C07321=1123.386,90.409,-56.038,-179.966,7.860,149.482
C07322=1123.381,90.658,-56.056,-179.965,7.864,149.482
C07323=1123.376,90.907,-56.074,-179.963,7.868,149.483
C07324=1123.371,91.156,-56.092,-179.961,7.872,149.483
C07325=1123.366,91.406,-56.111,-179.960,7.876,149.484
C07326=1123.362,91.655,-56.129,-179.958,7.879,149.484
C07327=1123.357,91.904,-56.147,-179.957,7.883,149.484
C07328=1123.352,92.153,-56.165,-179.956,7.886,149.485
C07329=1123.347,92.403,-56.183,-179.954,7.891,149.486
C07330=1123.343,92.652,-56.202,-179.953,7.895,149.486
C07331=1123.337,92.902,-56.220,-179.951,7.898,149.486
C07332=1123.332,93.150,-56.239,-179.950,7.902,149.487
C07333=1123.327,93.400,-56.257,-179.948,7.906,149.487
C07334=1123.323,93.650,-56.275,-179.946,7.910,149.488
C07335=1123.318,93.899,-56.293,-179.945,7.914,149.488
C07336=1123.313,94.148,-56.312,-179.943,7.918,149.489
C07337=1123.308,94.397,-56.331,-179.942,7.922,149.489
C07338=1123.304,94.647,-56.349,-179.939,7.926,149.489
C07339=1123.299,94.896,-56.367,-179.938,7.930,149.490
C07340=1123.293,95.145,-56.386,-179.936,7.934,149.490
C07341=1123.289,95.395,-56.404,-179.934,7.938,149.491
C07342=1123.284,95.644,-56.422,-179.933,7.942,149.491
C07343=1123.280,95.892,-56.441,-179.931,7.946,149.491
C07344=1123.274,96.142,-56.460,-179.929,7.949,149.492
C07345=1123.270,96.392,-56.478,-179.928,7.953,149.492
C07346=1123.265,96.640,-56.497,-179.926,7.957,149.493
C07347=1123.259,96.890,-56.515,-179.925,7.961,149.493
C07348=1123.255,97.140,-56.534,-179.923,7.965,149.493
C07349=1123.250,97.388,-56.552,-179.921,7.969,149.494
C07350=1123.245,97.638,-56.571,-179.919,7.973,149.494
C07351=1123.241,97.887,-56.590,-179.917,7.977,149.495
C07352=1123.236,98.136,-56.608,-179.916,7.981,149.495
C07353=1123.230,98.386,-56.627,-179.913,7.984,149.495
C07354=1123.226,98.635,-56.646,-179.912,7.988,149.496
C07355=1123.221,98.884,-56.664,-179.910,7.992,149.496
C07356=1123.216,99.133,-56.683,-179.908,7.997,149.497
C07357=1123.212,99.383,-56.701,-179.906,8.000,149.497
C07358=1123.206,99.632,-56.721,-179.904,8.004,149.497
C07359=1123.202,99.881,-56.739,-179.903,8.008,149.498
C07360=1123.197,100.130,-56.758,-179.901,8.012,149.498
C07361=1123.192,100.379,-56.777,-179.898,8.016,149.498
C07362=1123.188,100.629,-56.795,-179.896,8.020,149.498
C07363=1123.182,100.878,-56.815,-179.895,8.024,149.499
C07364=1123.178,101.127,-56.833,-179.893,8.028,149.499
C07365=1123.173,101.376,-56.852,-179.891,8.031,149.500
C07366=1123.168,101.626,-56.870,-179.889,8.036,149.500
C07367=1123.163,101.875,-56.890,-179.887,8.039,149.500
C07368=1123.158,102.124,-56.908,-179.885,8.043,149.501
C07369=1123.153,102.374,-56.927,-179.883,8.047,149.501
C07370=1123.150,102.588,-56.944,-179.882,8.051,149.501
C07371=1123.145,102.802,-56.960,-179.880,8.054,149.502
C07372=1123.141,103.016,-56.976,-179.878,8.058,149.502
C07373=1123.136,103.232,-56.992,-179.877,8.061,149.502
C07374=1123.133,103.446,-57.009,-179.874,8.064,149.502
C07375=1123.129,103.661,-57.025,-179.872,8.068,149.503
C07376=1123.125,103.875,-57.042,-179.871,8.070,149.503
C07377=1123.120,104.089,-57.058,-179.869,8.074,149.503
C07378=1123.115,104.339,-57.077,-179.867,8.078,149.503
C07379=1123.111,104.588,-57.096,-179.865,8.082,149.504
C07380=1123.106,104.838,-57.116,-179.863,8.086,149.504
C07381=1123.101,105.086,-57.134,-179.861,8.089,149.504
C07382=1123.096,105.336,-57.153,-179.858,8.094,149.505
C07383=1123.092,105.585,-57.172,-179.857,8.098,149.505
C07384=1123.087,105.834,-57.192,-179.855,8.101,149.505
C07385=1123.081,106.083,-57.211,-179.852,8.105,149.505
C07386=1123.077,106.333,-57.230,-179.850,8.109,149.506
C07387=1123.072,106.581,-57.249,-179.848,8.114,149.506
C07388=1123.067,106.831,-57.269,-179.846,8.117,149.506
C07389=1123.062,107.080,-57.287,-179.844,8.121,149.507
C07390=1123.058,107.330,-57.306,-179.841,8.125,149.507
C07391=1123.052,107.579,-57.326,-179.839,8.128,149.507
C07392=1123.048,107.828,-57.345,-179.837,8.132,149.507
C07393=1123.044,108.077,-57.364,-179.834,8.137,149.508
C07394=1123.038,108.326,-57.384,-179.832,8.140,149.508
C07395=1123.033,108.576,-57.403,-179.830,8.144,149.508
C07396=1123.029,108.824,-57.422,-179.828,8.148,149.508
C07397=1123.024,109.074,-57.442,-179.825,8.152,149.508
C07398=1123.019,109.324,-57.461,-179.823,8.156,149.509
C07399=1123.015,109.572,-57.480,-179.821,8.159,149.509
C07400=1123.010,109.822,-57.500,-179.818,8.163,149.509
C07401=1123.005,110.071,-57.519,-179.816,8.167,149.509
C07402=1123.000,110.320,-57.539,-179.813,8.171,149.510
C07403=1122.995,110.570,-57.558,-179.811,8.175,149.510
C07404=1122.991,110.818,-57.577,-179.809,8.179,149.510
C07405=1122.986,111.067,-57.597,-179.807,8.182,149.510
C07406=1122.981,111.317,-57.617,-179.805,8.186,149.510
C07407=1122.976,111.566,-57.636,-179.803,8.190,149.511
C07408=1122.971,111.815,-57.656,-179.801,8.193,149.511
C07409=1122.967,112.065,-57.676,-179.799,8.197,149.511
C07410=1122.962,112.313,-57.694,-179.797,8.200,149.512
C07411=1122.957,112.563,-57.714,-179.796,8.203,149.512
C07412=1122.953,112.812,-57.734,-179.794,8.207,149.512
C07413=1122.947,113.061,-57.754,-179.792,8.210,149.512
C07414=1122.943,113.310,-57.773,-179.790,8.214,149.513
C07415=1122.938,113.560,-57.793,-179.788,8.218,149.513
C07416=1122.933,113.809,-57.812,-179.786,8.221,149.513
C07417=1122.928,114.058,-57.833,-179.784,8.225,149.514
C07418=1122.923,114.307,-57.852,-179.782,8.228,149.514
C07419=1122.918,114.556,-57.872,-179.781,8.231,149.514
C07420=1122.913,114.806,-57.891,-179.779,8.235,149.514
C07421=1122.910,115.054,-57.911,-179.777,8.238,149.515
C07422=1122.905,115.304,-57.931,-179.775,8.242,149.515
C07423=1122.900,115.553,-57.950,-179.773,8.245,149.515
C07424=1122.895,115.802,-57.970,-179.771,8.249,149.516
C07425=1122.890,116.051,-57.990,-179.769,8.253,149.516
C07426=1122.886,116.266,-58.007,-179.767,8.256,149.516
C07427=1122.882,116.480,-58.025,-179.766,8.258,149.516
C07428=1122.878,116.695,-58.041,-179.765,8.261,149.516
C07429=1122.873,116.908,-58.059,-179.763,8.264,149.517
C07430=1122.869,117.123,-58.076,-179.761,8.267,149.517
C07431=1122.865,117.338,-58.092,-179.760,8.270,149.517
C07432=1122.861,117.552,-58.110,-179.758,8.273,149.517
C07433=1122.857,117.767,-58.127,-179.756,8.276,149.518
C07434=1122.852,118.016,-58.147,-179.755,8.280,149.518
C07435=1122.847,118.265,-58.167,-179.753,8.283,149.518
C07436=1122.842,118.514,-58.187,-179.751,8.286,149.518
C07437=1122.838,118.763,-58.207,-179.749,8.290,149.519
C07438=1122.833,119.012,-58.227,-179.747,8.293,149.519
C07439=1122.829,119.262,-58.247,-179.745,8.297,149.519
C07440=1122.824,119.511,-58.266,-179.744,8.300,149.520
C07441=1122.819,119.760,-58.287,-179.742,8.303,149.520
C07442=1122.814,120.008,-58.307,-179.740,8.307,149.520
C07443=1122.810,120.258,-58.326,-179.738,8.310,149.520
C07444=1122.805,120.507,-58.347,-179.737,8.313,149.521
C07445=1122.800,120.757,-58.366,-179.735,8.317,149.521
C07446=1122.796,121.005,-58.387,-179.733,8.320,149.521
C07447=1122.790,121.255,-58.407,-179.730,8.324,149.521
C07448=1122.785,121.504,-58.427,-179.729,8.327,149.522
C07449=1122.781,121.753,-58.447,-179.727,8.330,149.522
C07450=1122.776,122.002,-58.467,-179.725,8.334,149.522
C07451=1122.772,122.251,-58.487,-179.723,8.337,149.522
C07452=1122.767,122.501,-58.507,-179.722,8.340,149.523
C07453=1122.762,122.750,-58.528,-179.720,8.344,149.523
C07454=1122.757,122.999,-58.548,-179.718,8.348,149.523
C07455=1122.753,123.248,-58.568,-179.716,8.351,149.524
C07456=1122.748,123.497,-58.588,-179.715,8.354,149.524
C07457=1122.743,123.746,-58.608,-179.713,8.357,149.524
C07458=1122.738,123.995,-58.628,-179.711,8.361,149.524
C07459=1122.733,124.244,-58.649,-179.709,8.364,149.525
C07460=1122.729,124.493,-58.669,-179.707,8.367,149.525
C07461=1122.724,124.742,-58.690,-179.705,8.371,149.525
C07462=1122.720,124.992,-58.709,-179.704,8.375,149.526
C07463=1122.715,125.241,-58.730,-179.702,8.377,149.526
C07464=1122.710,125.490,-58.751,-179.700,8.381,149.526
C07465=1122.706,125.739,-58.771,-179.698,8.384,149.526
C07466=1122.701,125.989,-58.791,-179.697,8.388,149.527
C07467=1122.696,126.238,-58.812,-179.695,8.391,149.527
C07468=1122.691,126.487,-58.832,-179.693,8.395,149.527
C07469=1122.687,126.736,-58.852,-179.692,8.397,149.527
C07470=1122.682,126.985,-58.873,-179.690,8.401,149.528
C07471=1122.676,127.234,-58.893,-179.688,8.405,149.528
C07472=1122.672,127.483,-58.913,-179.686,8.407,149.528
C07473=1122.667,127.732,-58.933,-179.684,8.411,149.528
C07474=1122.662,127.981,-58.954,-179.682,8.414,149.529
C07475=1122.658,128.230,-58.975,-179.681,8.417,149.529
C07476=1122.653,128.479,-58.996,-179.679,8.421,149.529
C07477=1122.648,128.728,-59.016,-179.677,8.424,149.530
C07478=1122.644,128.977,-59.036,-179.676,8.427,149.530
C07479=1122.639,129.226,-59.057,-179.674,8.431,149.530
C07480=1122.634,129.475,-59.078,-179.672,8.434,149.530
C07481=1122.629,129.725,-59.097,-179.671,8.437,149.531
C07482=1122.625,129.940,-59.116,-179.669,8.440,149.531
C07483=1122.621,130.154,-59.134,-179.668,8.444,149.531
C07484=1122.617,130.368,-59.151,-179.666,8.446,149.532
C07485=1122.614,130.583,-59.169,-179.665,8.449,149.532
C07486=1122.609,130.797,-59.187,-179.663,8.452,149.532
C07487=1122.605,131.011,-59.205,-179.662,8.455,149.532
C07488=1122.601,131.226,-59.222,-179.660,8.457,149.532
C07489=1122.597,131.439,-59.240,-179.659,8.460,149.533
C07490=1122.592,131.689,-59.261,-179.657,8.464,149.533
C07491=1122.587,131.938,-59.281,-179.655,8.467,149.533
C07492=1122.582,132.187,-59.302,-179.654,8.470,149.534
C07493=1122.578,132.436,-59.322,-179.652,8.474,149.534
C07494=1122.573,132.686,-59.344,-179.651,8.477,149.534
C07495=1122.569,132.935,-59.364,-179.649,8.480,149.534
C07496=1122.564,133.183,-59.386,-179.646,8.484,149.535
C07497=1122.559,133.432,-59.406,-179.645,8.487,149.535
C07498=1122.554,133.682,-59.427,-179.643,8.490,149.535
C07499=1122.550,133.931,-59.448,-179.642,8.493,149.536
C07500=1122.545,134.180,-59.469,-179.640,8.497,149.536
C07501=1122.540,134.429,-59.489,-179.638,8.500,149.536
C07502=1122.535,134.678,-59.510,-179.637,8.503,149.536
C07503=1122.531,134.926,-59.531,-179.635,8.507,149.537
C07504=1122.526,135.176,-59.552,-179.634,8.510,149.537
C07505=1122.522,135.425,-59.573,-179.632,8.513,149.537
C07506=1122.517,135.675,-59.594,-179.630,8.517,149.538
C07507=1122.512,135.923,-59.614,-179.629,8.520,149.538
C07508=1122.507,136.172,-59.636,-179.627,8.524,149.538
C07509=1122.502,136.421,-59.657,-179.625,8.526,149.539
C07510=1122.498,136.670,-59.677,-179.623,8.530,149.539
C07511=1122.493,136.920,-59.698,-179.622,8.534,149.539
C07512=1122.489,137.169,-59.719,-179.620,8.536,149.539
C07513=1122.484,137.418,-59.740,-179.619,8.540,149.540
C07514=1122.479,137.667,-59.761,-179.617,8.543,149.540
C07515=1122.474,137.916,-59.782,-179.615,8.546,149.540
C07516=1122.469,138.165,-59.803,-179.614,8.550,149.541
C07517=1122.465,138.414,-59.824,-179.612,8.553,149.541
C07518=1122.460,138.664,-59.845,-179.610,8.557,149.541
C07519=1122.456,138.912,-59.867,-179.609,8.560,149.542
C07520=1122.451,139.161,-59.887,-179.607,8.564,149.542
C07521=1122.446,139.410,-59.909,-179.606,8.566,149.542
C07522=1122.441,139.659,-59.930,-179.604,8.570,149.543
C07523=1122.437,139.909,-59.951,-179.603,8.573,149.543
C07524=1122.432,140.157,-59.972,-179.601,8.576,149.543
C07525=1122.427,140.407,-59.993,-179.600,8.579,149.544
C07526=1122.423,140.655,-60.014,-179.598,8.583,149.544
C07527=1122.418,140.904,-60.035,-179.596,8.587,149.544
C07528=1122.413,141.154,-60.057,-179.595,8.589,149.545
C07529=1122.408,141.403,-60.078,-179.593,8.593,149.545
C07530=1122.404,141.652,-60.099,-179.592,8.596,149.545
C07531=1122.399,141.900,-60.120,-179.590,8.600,149.546
C07532=1122.395,142.150,-60.142,-179.589,8.603,149.546
C07533=1122.390,142.399,-60.163,-179.587,8.606,149.546
C07534=1122.385,142.648,-60.184,-179.586,8.610,149.547
C07535=1122.380,142.897,-60.205,-179.584,8.613,149.547
C07536=1122.376,143.147,-60.227,-179.583,8.616,149.547
C07537=1122.371,143.395,-60.248,-179.581,8.620,149.548
C07538=1122.367,143.610,-60.266,-179.580,8.623,149.548
C07539=1122.363,143.823,-60.285,-179.578,8.625,149.548
C07540=1122.359,144.038,-60.303,-179.577,8.628,149.549
C07541=1122.355,144.252,-60.322,-179.576,8.631,149.549
C07542=1122.351,144.466,-60.340,-179.574,8.634,149.549
C07543=1122.347,144.681,-60.359,-179.573,8.637,149.550
C07544=1122.343,144.895,-60.376,-179.572,8.640,149.550
C07545=1122.339,145.109,-60.395,-179.570,8.642,149.550
C07546=1122.334,145.359,-60.416,-179.568,8.647,149.550
C07547=1122.329,145.607,-60.438,-179.566,8.650,149.551
C07548=1122.324,145.856,-60.460,-179.563,8.654,149.551
C07549=1122.321,146.105,-60.481,-179.561,8.658,149.551
C07550=1122.316,146.354,-60.502,-179.558,8.662,149.551
C07551=1122.311,146.603,-60.524,-179.556,8.666,149.552
C07552=1122.306,146.853,-60.545,-179.553,8.670,149.552
C07553=1122.301,147.101,-60.567,-179.551,8.673,149.552
C07554=1122.297,147.350,-60.589,-179.548,8.677,149.552
C07555=1122.292,147.600,-60.610,-179.546,8.681,149.552
C07556=1122.287,147.849,-60.632,-179.543,8.685,149.552
C07557=1122.282,148.097,-60.653,-179.541,8.689,149.553
C07558=1122.278,148.347,-60.675,-179.538,8.693,149.553
C07559=1122.273,148.595,-60.697,-179.536,8.696,149.553
C07560=1122.268,148.844,-60.718,-179.533,8.700,149.553
C07561=1122.264,149.093,-60.740,-179.531,8.704,149.553
C07562=1122.260,149.342,-60.761,-179.529,8.707,149.554
C07563=1122.255,149.591,-60.783,-179.526,8.712,149.554
C07564=1122.250,149.840,-60.805,-179.524,8.715,149.554
C07565=1122.245,150.089,-60.827,-179.521,8.719,149.554
C07566=1122.240,150.339,-60.849,-179.519,8.722,149.554
C07567=1122.235,150.588,-60.870,-179.517,8.726,149.555
C07568=1122.231,150.837,-60.892,-179.514,8.730,149.555
C07569=1122.226,151.086,-60.914,-179.512,8.733,149.555
C07570=1122.222,151.335,-60.936,-179.510,8.737,149.555
C07571=1122.217,151.584,-60.958,-179.506,8.741,149.555
C07572=1122.212,151.832,-60.979,-179.504,8.744,149.555
C07573=1122.208,152.082,-61.001,-179.502,8.748,149.556
C07574=1122.203,152.330,-61.023,-179.499,8.751,149.556
C07575=1122.199,152.580,-61.045,-179.497,8.755,149.556
C07576=1122.194,152.828,-61.067,-179.495,8.758,149.556
C07577=1122.190,153.078,-61.089,-179.492,8.762,149.556
C07578=1122.184,153.327,-61.111,-179.490,8.766,149.556
C07579=1122.180,153.576,-61.133,-179.487,8.769,149.556
C07580=1122.175,153.824,-61.155,-179.485,8.772,149.557
C07581=1122.171,154.074,-61.177,-179.483,8.776,149.557
C07582=1122.166,154.322,-61.199,-179.480,8.780,149.557
C07583=1122.162,154.571,-61.221,-179.478,8.783,149.557
C07584=1122.156,154.820,-61.244,-179.475,8.786,149.557
C07585=1122.152,155.069,-61.266,-179.473,8.790,149.557
C07586=1122.147,155.318,-61.287,-179.471,8.793,149.557
C07587=1122.143,155.567,-61.309,-179.468,8.797,149.558
C07588=1122.138,155.816,-61.331,-179.465,8.800,149.558
C07589=1122.133,156.065,-61.354,-179.463,8.804,149.558
C07590=1122.129,156.314,-61.377,-179.461,8.807,149.558
C07591=1122.124,156.563,-61.398,-179.459,8.810,149.558
C07592=1122.120,156.812,-61.420,-179.456,8.814,149.558
C07593=1122.115,157.061,-61.443,-179.454,8.818,149.559
C07594=1122.111,157.275,-61.462,-179.452,8.820,149.559
C07595=1122.107,157.489,-61.481,-179.449,8.823,149.559
C07596=1122.103,157.703,-61.500,-179.448,8.826,149.559
C07597=1122.099,157.917,-61.519,-179.445,8.829,149.559
C07598=1122.095,158.131,-61.538,-179.444,8.832,149.559
C07599=1122.091,158.346,-61.557,-179.441,8.835,149.559
C07600=1122.087,158.560,-61.577,-179.439,8.837,149.559
C07601=1122.084,158.774,-61.596,-179.437,8.841,149.559
C07602=1122.078,159.023,-61.619,-179.435,8.844,149.559
C07603=1122.074,159.272,-61.641,-179.433,8.847,149.560
C07604=1122.069,159.520,-61.663,-179.430,8.850,149.560
C07605=1122.064,159.770,-61.686,-179.428,8.853,149.560
C07606=1122.060,160.019,-61.709,-179.425,8.857,149.560
C07607=1122.055,160.267,-61.730,-179.423,8.860,149.560
C07608=1122.050,160.517,-61.753,-179.421,8.864,149.560
C07609=1122.046,160.766,-61.776,-179.418,8.867,149.560
C07610=1122.041,161.014,-61.797,-179.416,8.870,149.560
C07611=1122.037,161.263,-61.821,-179.414,8.873,149.561
C07612=1122.032,161.513,-61.843,-179.411,8.876,149.561
C07613=1122.027,161.761,-61.866,-179.409,8.880,149.561
C07614=1122.023,162.010,-61.888,-179.407,8.883,149.561
C07615=1122.019,162.259,-61.911,-179.404,8.886,149.561
C07616=1122.014,162.509,-61.933,-179.402,8.890,149.561
C07617=1122.009,162.757,-61.956,-179.399,8.893,149.561
C07618=1122.004,163.006,-61.978,-179.397,8.896,149.561
C07619=1122.000,163.255,-62.001,-179.395,8.899,149.561
C07620=1121.995,163.504,-62.024,-179.392,8.902,149.561
C07621=1121.991,163.753,-62.046,-179.390,8.905,149.561
C07622=1121.986,164.002,-62.069,-179.388,8.909,149.562
C07623=1121.982,164.251,-62.091,-179.385,8.912,149.562
C07624=1121.977,164.500,-62.114,-179.383,8.915,149.562
C07625=1121.973,164.748,-62.137,-179.381,8.919,149.562
C07626=1121.968,164.998,-62.160,-179.378,8.922,149.562
C07627=1121.964,165.247,-62.183,-179.376,8.924,149.562
C07628=1121.958,165.495,-62.206,-179.374,8.928,149.562
C07629=1121.954,165.744,-62.228,-179.372,8.931,149.562
C07630=1121.949,165.993,-62.251,-179.369,8.934,149.562
C07631=1121.945,166.242,-62.274,-179.367,8.937,149.563
C07632=1121.940,166.490,-62.297,-179.364,8.940,149.563
C07633=1121.935,166.740,-62.319,-179.362,8.944,149.563
C07634=1121.931,166.989,-62.342,-179.359,8.947,149.563
C07635=1121.926,167.238,-62.366,-179.358,8.949,149.563
C07636=1121.922,167.487,-62.389,-179.355,8.952,149.563
C07637=1121.917,167.736,-62.411,-179.353,8.956,149.563
C07638=1121.912,167.985,-62.434,-179.351,8.959,149.563
C07639=1121.908,168.233,-62.457,-179.348,8.962,149.563
C07640=1121.903,168.482,-62.480,-179.346,8.965,149.563
C07641=1121.899,168.731,-62.503,-179.344,8.968,149.564
C07642=1121.894,168.979,-62.526,-179.342,8.971,149.564
C07643=1121.889,169.229,-62.548,-179.339,8.974,149.564
C07644=1121.885,169.478,-62.572,-179.337,8.977,149.564
C07645=1121.880,169.727,-62.595,-179.335,8.981,149.564
C07646=1121.876,169.976,-62.618,-179.333,8.983,149.564
C07647=1121.871,170.225,-62.641,-179.330,8.986,149.564
C07648=1121.866,170.473,-62.664,-179.328,8.990,149.564
C07649=1121.862,170.722,-62.687,-179.326,8.993,149.564
C07650=1121.858,170.936,-62.708,-179.324,8.995,149.564
C07651=1121.854,171.151,-62.727,-179.322,8.997,149.564
C07652=1121.850,171.364,-62.747,-179.320,9.000,149.565
C07653=1121.846,171.578,-62.767,-179.318,9.003,149.565
C07654=1121.842,171.792,-62.787,-179.316,9.006,149.565
C07655=1121.838,172.007,-62.806,-179.314,9.008,149.565
C07656=1121.834,172.220,-62.827,-179.313,9.011,149.565
C07657=1121.830,172.434,-62.847,-179.310,9.014,149.565
C07658=1121.825,172.683,-62.870,-179.308,9.016,149.565
C07659=1121.821,172.932,-62.893,-179.306,9.019,149.565
C07660=1121.817,173.181,-62.916,-179.304,9.023,149.565
C07661=1121.812,173.430,-62.939,-179.302,9.025,149.565
C07662=1121.807,173.679,-62.963,-179.299,9.028,149.565
C07663=1121.803,173.928,-62.986,-179.297,9.032,149.566
C07664=1121.798,174.177,-63.009,-179.295,9.035,149.566
C07665=1121.793,174.426,-63.033,-179.293,9.037,149.566
C07666=1121.790,174.674,-63.056,-179.290,9.040,149.566
C07667=1121.785,174.923,-63.080,-179.288,9.044,149.566
C07668=1121.780,175.172,-63.103,-179.286,9.046,149.566
C07669=1121.775,175.421,-63.126,-179.284,9.049,149.566
C07670=1121.771,175.670,-63.150,-179.282,9.053,149.566
C07671=1121.766,175.919,-63.173,-179.280,9.055,149.566
C07672=1121.762,176.168,-63.197,-179.277,9.058,149.566
C07673=1121.758,176.416,-63.220,-179.275,9.061,149.566
C07674=1121.753,176.665,-63.243,-179.273,9.064,149.567
C07675=1121.748,176.914,-63.267,-179.271,9.067,149.567
C07676=1121.744,177.163,-63.291,-179.269,9.070,149.567
C07677=1121.739,177.412,-63.314,-179.267,9.073,149.567
C07678=1121.734,177.661,-63.337,-179.264,9.076,149.567
C07679=1121.730,177.910,-63.361,-179.263,9.079,149.567
C07680=1121.725,178.158,-63.385,-179.260,9.082,149.567
C07681=1121.721,178.407,-63.408,-179.258,9.085,149.567
C07682=1121.716,178.656,-63.432,-179.256,9.087,149.567
C07683=1121.712,178.905,-63.456,-179.254,9.091,149.567
C07684=1121.707,179.154,-63.479,-179.252,9.093,149.568
C07685=1121.702,179.403,-63.502,-179.249,9.097,149.568
C07686=1121.698,179.651,-63.526,-179.246,9.100,149.568
C07687=1121.693,179.900,-63.550,-179.244,9.103,149.568
C07688=1121.688,180.149,-63.573,-179.241,9.106,149.568
C07689=1121.684,180.398,-63.597,-179.238,9.110,149.568
C07690=1121.679,180.647,-63.621,-179.235,9.113,149.568
C07691=1121.675,180.895,-63.645,-179.233,9.116,149.568
C07692=1121.670,181.144,-63.668,-179.230,9.119,149.568
C07693=1121.666,181.393,-63.692,-179.227,9.123,149.568
C07694=1121.662,181.642,-63.716,-179.224,9.126,149.568
C07695=1121.657,181.891,-63.740,-179.222,9.129,149.568
C07696=1121.653,182.140,-63.763,-179.219,9.132,149.568
C07697=1121.648,182.388,-63.787,-179.216,9.135,149.568
C07698=1121.644,182.637,-63.811,-179.214,9.138,149.568
C07699=1121.639,182.886,-63.835,-179.211,9.141,149.568
C07700=1121.634,183.135,-63.859,-179.209,9.144,149.568
C07701=1121.629,183.383,-63.883,-179.206,9.147,149.568
C07702=1121.625,183.632,-63.906,-179.204,9.150,149.568
C07703=1121.621,183.882,-63.931,-179.201,9.154,149.568
C07704=1121.616,184.130,-63.955,-179.198,9.156,149.568
C07705=1121.612,184.379,-63.978,-179.196,9.159,149.568
C07706=1121.608,184.592,-63.999,-179.193,9.162,149.568
C07707=1121.604,184.807,-64.020,-179.191,9.165,149.568
C07708=1121.600,185.020,-64.040,-179.189,9.167,149.568
C07709=1121.596,185.234,-64.061,-179.187,9.170,149.568
C07710=1121.592,185.448,-64.082,-179.185,9.173,149.568
C07711=1121.588,185.663,-64.102,-179.183,9.175,149.568
C07712=1121.584,185.876,-64.123,-179.180,9.178,149.568
C07713=1121.580,186.090,-64.144,-179.178,9.180,149.568
C07714=1121.576,186.339,-64.168,-179.176,9.183,149.568
C07715=1121.572,186.587,-64.192,-179.174,9.185,149.568
C07716=1121.566,186.837,-64.216,-179.171,9.189,149.568
C07717=1121.562,187.086,-64.240,-179.169,9.192,149.568
C07718=1121.558,187.334,-64.264,-179.167,9.194,149.568
C07719=1121.553,187.583,-64.289,-179.164,9.197,149.568
C07720=1121.548,187.832,-64.312,-179.162,9.200,149.568
C07721=1121.544,188.080,-64.336,-179.160,9.203,149.568
C07722=1121.540,188.329,-64.361,-179.157,9.206,149.568
C07723=1121.535,188.578,-64.385,-179.155,9.209,149.568
C07724=1121.530,188.826,-64.410,-179.153,9.211,149.568
C07725=1121.526,189.075,-64.434,-179.150,9.214,149.568
C07726=1121.521,189.325,-64.458,-179.148,9.217,149.568
C07727=1121.517,189.573,-64.482,-179.146,9.220,149.569
C07728=1121.512,189.822,-64.506,-179.144,9.222,149.569
C07729=1121.507,190.070,-64.531,-179.141,9.225,149.569
C07730=1121.504,190.320,-64.555,-179.140,9.227,149.569
C07731=1121.498,190.568,-64.580,-179.137,9.230,149.569
C07732=1121.494,190.817,-64.604,-179.135,9.233,149.569
C07733=1121.490,191.066,-64.628,-179.133,9.236,149.569
C07734=1121.485,191.315,-64.653,-179.131,9.239,149.569
C07735=1121.481,191.563,-64.677,-179.129,9.242,149.569
C07736=1121.476,191.812,-64.702,-179.127,9.244,149.569
C07737=1121.472,192.061,-64.726,-179.125,9.246,149.569
C07738=1121.467,192.309,-64.750,-179.122,9.250,149.569
C07739=1121.462,192.558,-64.775,-179.121,9.252,149.569
C07740=1121.458,192.807,-64.799,-179.119,9.255,149.569
C07741=1121.453,193.056,-64.824,-179.116,9.258,149.569
C07742=1121.449,193.304,-64.848,-179.115,9.260,149.570
C07743=1121.444,193.554,-64.873,-179.113,9.263,149.570
C07744=1121.440,193.802,-64.897,-179.111,9.265,149.570
C07745=1121.435,194.051,-64.922,-179.109,9.268,149.570
C07746=1121.431,194.300,-64.946,-179.107,9.271,149.570
C07747=1121.426,194.549,-64.971,-179.105,9.273,149.570
C07748=1121.422,194.797,-64.995,-179.104,9.276,149.570
C07749=1121.418,195.046,-65.020,-179.101,9.279,149.570
C07750=1121.413,195.294,-65.045,-179.100,9.282,149.571
C07751=1121.409,195.543,-65.069,-179.098,9.284,149.571
C07752=1121.404,195.792,-65.094,-179.096,9.287,149.571
C07753=1121.399,196.041,-65.119,-179.095,9.289,149.571
C07754=1121.395,196.290,-65.143,-179.093,9.292,149.571
C07755=1121.390,196.539,-65.168,-179.090,9.296,149.571
C07756=1121.386,196.787,-65.192,-179.086,9.299,149.571
C07757=1121.381,197.036,-65.218,-179.083,9.303,149.571
C07758=1121.377,197.284,-65.242,-179.080,9.307,149.571
C07759=1121.372,197.534,-65.267,-179.077,9.309,149.571
C07760=1121.368,197.782,-65.291,-179.073,9.313,149.571
C07761=1121.363,198.030,-65.316,-179.070,9.317,149.571
C07762=1121.360,198.244,-65.338,-179.067,9.319,149.571
C07763=1121.356,198.458,-65.359,-179.064,9.322,149.571
C07764=1121.352,198.673,-65.380,-179.061,9.325,149.571
C07765=1121.348,198.886,-65.401,-179.059,9.328,149.570
C07766=1121.344,199.100,-65.423,-179.056,9.331,149.570
C07767=1121.341,199.314,-65.444,-179.053,9.334,149.570
C07768=1121.336,199.527,-65.465,-179.050,9.337,149.570
C07769=1121.332,199.741,-65.487,-179.047,9.339,149.570
C07770=1121.329,199.990,-65.512,-179.045,9.342,149.570
C07771=1121.323,200.239,-65.537,-179.041,9.346,149.570
C07772=1121.319,200.487,-65.563,-179.038,9.349,149.570
C07773=1121.315,200.736,-65.587,-179.035,9.352,149.570
C07774=1121.310,200.985,-65.612,-179.032,9.355,149.570
C07775=1121.305,201.233,-65.637,-179.028,9.358,149.569
C07776=1121.302,201.482,-65.662,-179.025,9.362,149.569
C07777=1121.297,201.731,-65.687,-179.023,9.364,149.569
C07778=1121.292,201.980,-65.712,-179.019,9.368,149.569
C07779=1121.287,202.228,-65.738,-179.016,9.371,149.569
C07780=1121.284,202.477,-65.763,-179.013,9.373,149.569
C07781=1121.279,202.725,-65.787,-179.009,9.377,149.569
C07782=1121.275,202.974,-65.813,-179.007,9.380,149.569
C07783=1121.269,203.223,-65.838,-179.004,9.383,149.569
C07784=1121.265,203.472,-65.864,-179.001,9.385,149.568
C07785=1121.261,203.721,-65.888,-178.997,9.389,149.568
C07786=1121.257,203.969,-65.913,-178.994,9.392,149.568
C07787=1121.252,204.218,-65.939,-178.992,9.395,149.568
C07788=1121.247,204.466,-65.964,-178.989,9.398,149.568
C07789=1121.243,204.715,-65.990,-178.986,9.400,149.568
C07790=1121.238,204.963,-66.015,-178.983,9.403,149.568
C07791=1121.234,205.213,-66.040,-178.981,9.406,149.568
C07792=1121.229,205.462,-66.066,-178.978,9.409,149.568
C07793=1121.225,205.709,-66.090,-178.975,9.412,149.568
C07794=1121.221,205.958,-66.116,-178.972,9.414,149.567
C07795=1121.216,206.207,-66.141,-178.969,9.417,149.567
C07796=1121.212,206.456,-66.167,-178.966,9.420,149.567
C07797=1121.208,206.704,-66.192,-178.964,9.423,149.567
C07798=1121.203,206.953,-66.218,-178.961,9.426,149.567
C07799=1121.199,207.201,-66.244,-178.958,9.429,149.567
C07800=1121.194,207.451,-66.269,-178.955,9.432,149.567
C07801=1121.189,207.699,-66.294,-178.952,9.435,149.567
C07802=1121.185,207.948,-66.320,-178.950,9.438,149.567
C07803=1121.181,208.196,-66.345,-178.947,9.440,149.567
C07804=1121.176,208.445,-66.371,-178.945,9.443,149.567
C07805=1121.172,208.693,-66.397,-178.942,9.446,149.567
C07806=1121.167,208.942,-66.422,-178.939,9.449,149.567
C07807=1121.163,209.190,-66.448,-178.937,9.451,149.567
C07808=1121.158,209.440,-66.473,-178.935,9.454,149.567
C07809=1121.154,209.689,-66.499,-178.932,9.457,149.567
C07810=1121.149,209.937,-66.524,-178.929,9.460,149.567
C07811=1121.145,210.185,-66.550,-178.927,9.463,149.567
C07812=1121.141,210.434,-66.575,-178.925,9.465,149.567
C07813=1121.136,210.683,-66.601,-178.922,9.468,149.567
C07814=1121.132,210.931,-66.627,-178.919,9.471,149.567
C07815=1121.127,211.180,-66.652,-178.917,9.473,149.567
C07816=1121.122,211.429,-66.679,-178.915,9.476,149.567
C07817=1121.118,211.678,-66.704,-178.912,9.479,149.567
C07818=1121.114,211.890,-66.726,-178.910,9.482,149.567
C07819=1121.110,212.104,-66.749,-178.909,9.484,149.567
C07820=1121.107,212.318,-66.770,-178.907,9.486,149.567
C07821=1121.103,212.532,-66.793,-178.905,9.489,149.567
C07822=1121.099,212.746,-66.815,-178.903,9.491,149.567
C07823=1121.096,212.959,-66.837,-178.901,9.493,149.567
C07824=1121.092,213.173,-66.860,-178.899,9.496,149.567
C07825=1121.088,213.387,-66.881,-178.898,9.498,149.567
C07826=1121.083,213.636,-66.908,-178.895,9.502,149.568
C07827=1121.079,213.884,-66.934,-178.893,9.504,149.568
C07828=1121.074,214.132,-66.959,-178.891,9.507,149.568
C07829=1121.070,214.381,-66.985,-178.889,9.510,149.568
C07830=1121.066,214.630,-67.011,-178.887,9.512,149.568
C07831=1121.061,214.879,-67.037,-178.885,9.516,149.568
C07832=1121.057,215.128,-67.063,-178.883,9.518,149.568
C07833=1121.052,215.375,-67.089,-178.881,9.521,149.568
C07834=1121.048,215.624,-67.115,-178.879,9.524,149.569
C07835=1121.044,215.873,-67.141,-178.877,9.527,149.569
C07836=1121.039,216.122,-67.167,-178.875,9.530,149.569
C07837=1121.035,216.370,-67.193,-178.873,9.533,149.569
C07838=1121.031,216.619,-67.219,-178.870,9.536,149.569
C07839=1121.026,216.867,-67.245,-178.868,9.539,149.569
C07840=1121.021,217.116,-67.271,-178.866,9.541,149.569
C07841=1121.017,217.364,-67.297,-178.864,9.545,149.569
C07842=1121.013,217.613,-67.323,-178.861,9.548,149.569
C07843=1121.008,217.862,-67.349,-178.860,9.550,149.570
C07844=1121.004,218.110,-67.376,-178.857,9.554,149.570
C07845=1121.000,218.359,-67.402,-178.855,9.557,149.570
C07846=1120.995,218.607,-67.427,-178.852,9.560,149.570
C07847=1120.990,218.856,-67.454,-178.850,9.563,149.570
C07848=1120.986,219.104,-67.480,-178.848,9.566,149.570
C07849=1120.982,219.353,-67.506,-178.846,9.569,149.570
C07850=1120.978,219.601,-67.532,-178.843,9.572,149.570
C07851=1120.973,219.851,-67.558,-178.841,9.575,149.570
C07852=1120.969,220.099,-67.585,-178.838,9.578,149.570
C07853=1120.964,220.348,-67.611,-178.836,9.581,149.570
C07854=1120.960,220.596,-67.638,-178.833,9.585,149.571
C07855=1120.956,220.845,-67.663,-178.831,9.588,149.571
C07856=1120.950,221.093,-67.690,-178.828,9.591,149.571
C07857=1120.946,221.341,-67.716,-178.826,9.594,149.571
C07858=1120.942,221.590,-67.743,-178.823,9.597,149.571
C07859=1120.937,221.839,-67.769,-178.821,9.600,149.571
C07860=1120.933,222.087,-67.795,-178.818,9.603,149.571
C07861=1120.928,222.336,-67.822,-178.816,9.606,149.571
C07862=1120.925,222.584,-67.848,-178.813,9.609,149.571
C07863=1120.920,222.833,-67.874,-178.811,9.613,149.571
C07864=1120.916,223.082,-67.901,-178.807,9.616,149.571
C07865=1120.911,223.330,-67.928,-178.805,9.619,149.571
C07866=1120.907,223.579,-67.954,-178.802,9.622,149.571
C07867=1120.902,223.827,-67.981,-178.800,9.625,149.571
C07868=1120.898,224.076,-68.007,-178.797,9.629,149.571
C07869=1120.893,224.325,-68.034,-178.794,9.632,149.572
C07870=1120.889,224.573,-68.060,-178.791,9.635,149.571
C07871=1120.885,224.821,-68.087,-178.788,9.638,149.571
C07872=1120.880,225.070,-68.113,-178.786,9.641,149.572
C07873=1120.876,225.319,-68.140,-178.782,9.645,149.571
C07874=1120.872,225.532,-68.163,-178.780,9.647,149.571
C07875=1120.868,225.746,-68.185,-178.778,9.650,149.572
C07876=1120.865,225.959,-68.208,-178.775,9.653,149.571
C07877=1120.861,226.173,-68.232,-178.772,9.656,149.571
C07878=1120.857,226.387,-68.254,-178.770,9.659,149.572
C07879=1120.853,226.600,-68.277,-178.768,9.661,149.571
C07880=1120.849,226.813,-68.301,-178.765,9.664,149.571
C07881=1120.845,227.027,-68.323,-178.762,9.667,149.571
C07882=1120.841,227.275,-68.350,-178.759,9.670,149.571
C07883=1120.837,227.524,-68.377,-178.756,9.674,149.571
C07884=1120.833,227.772,-68.403,-178.753,9.677,149.571
C07885=1120.828,228.021,-68.430,-178.750,9.680,149.571
C07886=1120.824,228.270,-68.457,-178.747,9.683,149.571
C07887=1120.820,228.518,-68.484,-178.744,9.687,149.571
C07888=1120.815,228.767,-68.511,-178.741,9.690,149.571
C07889=1120.811,229.015,-68.538,-178.737,9.693,149.571
C07890=1120.807,229.264,-68.564,-178.734,9.696,149.571
C07891=1120.802,229.512,-68.591,-178.731,9.700,149.571
C07892=1120.797,229.761,-68.618,-178.728,9.702,149.571
C07893=1120.793,230.009,-68.645,-178.724,9.706,149.570
C07894=1120.789,230.257,-68.672,-178.721,9.709,149.570
C07895=1120.785,230.506,-68.699,-178.718,9.712,149.570
C07896=1120.780,230.755,-68.726,-178.715,9.715,149.570
C07897=1120.775,231.003,-68.753,-178.711,9.719,149.570
C07898=1120.772,231.252,-68.780,-178.709,9.721,149.570
C07899=1120.767,231.500,-68.807,-178.705,9.725,149.570
C07900=1120.762,231.749,-68.834,-178.702,9.728,149.570
C07901=1120.759,231.997,-68.862,-178.699,9.730,149.570
C07902=1120.754,232.246,-68.889,-178.695,9.734,149.570
C07903=1120.750,232.494,-68.916,-178.693,9.737,149.569
C07904=1120.745,232.742,-68.943,-178.690,9.739,149.569
C07905=1120.741,232.991,-68.970,-178.687,9.742,149.569
C07906=1120.737,233.240,-68.997,-178.684,9.745,149.569
C07907=1120.732,233.488,-69.025,-178.681,9.748,149.569
C07908=1120.728,233.736,-69.052,-178.677,9.751,149.569
C07909=1120.723,233.985,-69.079,-178.674,9.754,149.569
C07910=1120.720,234.234,-69.106,-178.671,9.757,149.569
C07911=1120.715,234.482,-69.134,-178.668,9.760,149.568
C07912=1120.711,234.730,-69.161,-178.665,9.762,149.568
C07913=1120.706,234.979,-69.188,-178.662,9.765,149.568
C07914=1120.702,235.228,-69.215,-178.660,9.768,149.568
C07915=1120.698,235.476,-69.243,-178.657,9.771,149.568
C07916=1120.693,235.724,-69.270,-178.655,9.773,149.568
C07917=1120.688,235.973,-69.297,-178.652,9.776,149.568
C07918=1120.684,236.221,-69.325,-178.649,9.778,149.568
C07919=1120.680,236.470,-69.352,-178.646,9.781,149.568
C07920=1120.675,236.718,-69.380,-178.643,9.784,149.568
C07921=1120.671,236.967,-69.408,-178.640,9.787,149.567
C07922=1120.667,237.215,-69.435,-178.638,9.789,149.567
C07923=1120.662,237.463,-69.462,-178.635,9.792,149.567
C07924=1120.658,237.712,-69.490,-178.632,9.794,149.567
C07925=1120.654,237.960,-69.518,-178.630,9.796,149.567
C07926=1120.647,238.351,-69.560,-178.626,9.801,149.567
C07927=1120.640,238.744,-69.604,-178.621,9.805,149.567
C07928=1120.633,239.136,-69.648,-178.618,9.809,149.567
C07929=1120.627,239.526,-69.691,-178.614,9.813,149.567
C07930=1120.622,239.811,-69.723,-178.611,9.816,149.567
C07931=1120.617,240.094,-69.754,-178.608,9.818,149.566
C07932=1120.612,240.378,-69.786,-178.605,9.821,149.567
C07933=1120.607,240.661,-69.817,-178.602,9.824,149.566
C07934=1120.603,240.910,-69.845,-178.600,9.827,149.566
C07935=1120.598,241.158,-69.872,-178.597,9.829,149.566
C07936=1120.593,241.407,-69.901,-178.596,9.832,149.566
C07937=1120.589,241.656,-69.928,-178.593,9.834,149.566
C07938=1120.585,241.904,-69.956,-178.591,9.837,149.566
C07939=1120.581,242.152,-69.984,-178.588,9.839,149.566
C07940=1120.576,242.401,-70.011,-178.586,9.841,149.566
C07941=1120.572,242.649,-70.039,-178.585,9.843,149.566
C07942=1120.568,242.897,-70.067,-178.582,9.846,149.566
C07943=1120.563,243.145,-70.096,-178.580,9.848,149.566
C07944=1120.559,243.395,-70.123,-178.578,9.851,149.566
C07945=1120.555,243.642,-70.151,-178.576,9.853,149.566
C07946=1120.550,243.890,-70.179,-178.574,9.855,149.566
C07947=1120.546,244.139,-70.206,-178.571,9.858,149.566
C07948=1120.541,244.388,-70.234,-178.569,9.860,149.566
C07949=1120.538,244.636,-70.262,-178.567,9.863,149.566
C07950=1120.533,244.884,-70.290,-178.565,9.865,149.567
C07951=1120.529,245.133,-70.318,-178.564,9.867,149.567
C07952=1120.525,245.381,-70.345,-178.562,9.870,149.567
C07953=1120.520,245.630,-70.374,-178.560,9.872,149.567
C07954=1120.516,245.878,-70.402,-178.558,9.874,149.567
C07955=1120.512,246.126,-70.430,-178.556,9.877,149.567
C07956=1120.507,246.375,-70.458,-178.554,9.880,149.567
C07957=1120.502,246.623,-70.486,-178.553,9.882,149.567
C07958=1120.499,246.872,-70.514,-178.551,9.884,149.567
C07959=1120.494,247.120,-70.541,-178.549,9.887,149.567
C07960=1120.490,247.369,-70.570,-178.547,9.889,149.568
C07961=1120.486,247.616,-70.598,-178.544,9.893,149.567
C07962=1120.482,247.865,-70.626,-178.538,9.897,149.567
C07963=1120.477,248.113,-70.654,-178.533,9.902,149.567
C07964=1120.473,248.362,-70.683,-178.528,9.905,149.566
C07965=1120.469,248.610,-70.710,-178.523,9.910,149.566
C07966=1120.464,248.858,-70.739,-178.518,9.914,149.566
C07967=1120.460,249.106,-70.767,-178.513,9.918,149.565
C07968=1120.456,249.355,-70.795,-178.508,9.922,149.565
C07969=1120.452,249.604,-70.824,-178.504,9.925,149.565
C07970=1120.447,249.852,-70.852,-178.500,9.929,149.564
C07971=1120.443,250.101,-70.880,-178.496,9.932,149.564
C07972=1120.438,250.348,-70.908,-178.492,9.935,149.564
C07973=1120.434,250.597,-70.937,-178.488,9.938,149.564
C07974=1120.430,250.846,-70.965,-178.484,9.941,149.563
C07975=1120.425,251.094,-70.993,-178.481,9.944,149.563
C07976=1120.422,251.342,-71.022,-178.477,9.947,149.563
C07977=1120.416,251.590,-71.051,-178.473,9.950,149.563
C07978=1120.413,251.839,-71.079,-178.470,9.953,149.562
C07979=1120.408,252.088,-71.107,-178.467,9.955,149.562
C07980=1120.404,252.335,-71.136,-178.464,9.958,149.562
C07981=1120.400,252.584,-71.165,-178.462,9.960,149.562
C07982=1120.396,252.797,-71.188,-178.459,9.962,149.562
C07983=1120.392,253.010,-71.213,-178.457,9.964,149.562
C07984=1120.389,253.224,-71.238,-178.455,9.966,149.562
C07985=1120.385,253.437,-71.262,-178.454,9.967,149.562
C07986=1120.382,253.650,-71.287,-178.452,9.969,149.562
C07987=1120.378,253.864,-71.312,-178.450,9.971,149.561
C07988=1120.374,254.077,-71.336,-178.449,9.972,149.561
C07989=1120.370,254.291,-71.360,-178.448,9.974,149.561
C07990=1120.366,254.538,-71.389,-178.445,9.976,149.561
C07991=1120.362,254.787,-71.418,-178.444,9.978,149.562
C07992=1120.357,255.036,-71.446,-178.443,9.979,149.562
C07993=1120.353,255.283,-71.475,-178.442,9.981,149.562
C07994=1120.349,255.532,-71.504,-178.442,9.982,149.562
C07995=1120.345,255.780,-71.532,-178.440,9.983,149.562
C07996=1120.340,256.028,-71.561,-178.439,9.985,149.562
C07997=1120.336,256.277,-71.590,-178.437,9.988,149.562
C07998=1120.332,256.525,-71.618,-178.434,9.991,149.562
C07999=1120.328,256.774,-71.647,-178.431,9.994,149.562
C08000=1120.323,257.021,-71.676,-178.428,9.997,149.562
C08001=1120.319,257.270,-71.704,-178.425,10.000,149.562
C08002=1120.315,257.519,-71.733,-178.422,10.002,149.562
C08003=1120.310,257.766,-71.762,-178.420,10.005,149.562
C08004=1120.306,258.015,-71.790,-178.417,10.008,149.562
C08005=1120.302,258.263,-71.820,-178.414,10.011,149.562
C08006=1120.298,258.512,-71.849,-178.411,10.014,149.561
C08007=1120.294,258.759,-71.877,-178.408,10.016,149.561
C08008=1120.289,259.008,-71.906,-178.405,10.019,149.561
C08009=1120.285,259.256,-71.935,-178.402,10.022,149.561
C08010=1120.280,259.505,-71.964,-178.399,10.025,149.561
C08011=1120.276,259.753,-71.992,-178.396,10.028,149.561
C08012=1120.272,260.001,-72.022,-178.393,10.031,149.561
C08013=1120.268,260.250,-72.051,-178.390,10.034,149.561
C08014=1120.264,260.498,-72.080,-178.387,10.036,149.561
C08015=1120.260,260.745,-72.109,-178.384,10.039,149.561
C08016=1120.255,260.994,-72.137,-178.380,10.042,149.560
C08017=1120.251,261.242,-72.167,-178.377,10.045,149.560
C08018=1120.247,261.491,-72.196,-178.374,10.048,149.560
C08019=1120.242,261.740,-72.225,-178.370,10.051,149.560
C08020=1120.239,261.988,-72.254,-178.367,10.054,149.560
C08021=1120.234,262.235,-72.283,-178.364,10.057,149.560
C08022=1120.229,262.484,-72.312,-178.361,10.060,149.559
C08023=1120.225,262.732,-72.341,-178.358,10.063,149.559
C08024=1120.221,262.981,-72.371,-178.354,10.065,149.559
C08025=1120.217,263.229,-72.400,-178.351,10.069,149.559
C08026=1120.212,263.478,-72.429,-178.347,10.071,149.559
C08027=1120.208,263.725,-72.457,-178.344,10.074,149.559
C08028=1120.204,263.973,-72.487,-178.340,10.077,149.558
C08029=1120.200,264.221,-72.516,-178.337,10.080,149.558
C08030=1120.196,264.470,-72.546,-178.333,10.083,149.558
C08031=1120.192,264.718,-72.575,-178.331,10.085,149.558
C08032=1120.187,264.966,-72.605,-178.328,10.088,149.558
C08033=1120.183,265.215,-72.633,-178.326,10.090,149.558
C08034=1120.179,265.463,-72.663,-178.323,10.093,149.557
C08035=1120.174,265.711,-72.692,-178.320,10.095,149.557
C08036=1120.170,265.959,-72.721,-178.318,10.097,149.557
C08037=1120.166,266.208,-72.751,-178.315,10.100,149.557
C08038=1120.162,266.421,-72.776,-178.312,10.102,149.557
C08039=1120.159,266.634,-72.802,-178.311,10.104,149.557
C08040=1120.155,266.847,-72.827,-178.308,10.106,149.557
C08041=1120.151,267.060,-72.852,-178.306,10.108,149.557
C08042=1120.148,267.273,-72.877,-178.304,10.110,149.557
C08043=1120.144,267.487,-72.902,-178.301,10.112,149.557
C08044=1120.141,267.700,-72.928,-178.299,10.115,149.557
C08045=1120.137,267.913,-72.953,-178.296,10.117,149.557
C08046=1120.133,268.161,-72.983,-178.294,10.119,149.556
C08047=1120.129,268.409,-73.012,-178.291,10.122,149.556
C08048=1120.125,268.658,-73.042,-178.288,10.125,149.556
C08049=1120.120,268.906,-73.072,-178.286,10.127,149.556
C08050=1120.116,269.155,-73.101,-178.283,10.130,149.556
C08051=1120.111,269.402,-73.130,-178.280,10.132,149.556
C08052=1120.107,269.650,-73.160,-178.278,10.134,149.556
C08053=1120.103,269.898,-73.190,-178.275,10.137,149.556
C08054=1120.098,270.146,-73.219,-178.272,10.140,149.556
C08055=1120.094,270.395,-73.249,-178.269,10.143,149.555
C08056=1120.090,270.643,-73.278,-178.266,10.145,149.555
C08057=1120.086,270.891,-73.308,-178.264,10.147,149.555
C08058=1120.081,271.140,-73.338,-178.261,10.150,149.555
C08059=1120.078,271.388,-73.368,-178.258,10.153,149.555
C08060=1120.074,271.636,-73.398,-178.255,10.156,149.555
C08061=1120.069,271.885,-73.427,-178.252,10.158,149.555
C08062=1120.065,272.133,-73.457,-178.249,10.161,149.555
C08063=1120.061,272.380,-73.487,-178.246,10.163,149.554
C08064=1120.056,272.629,-73.517,-178.243,10.166,149.554
C08065=1120.052,272.877,-73.546,-178.240,10.168,149.554
C08066=1120.048,273.125,-73.576,-178.238,10.171,149.554
C08067=1120.044,273.373,-73.606,-178.235,10.174,149.554
C08068=1120.040,273.622,-73.635,-178.232,10.177,149.554
C08069=1120.035,273.869,-73.666,-178.229,10.179,149.554
C08070=1120.031,274.118,-73.696,-178.226,10.182,149.554
C08071=1120.027,274.366,-73.725,-178.222,10.185,149.553
C08072=1120.023,274.614,-73.755,-178.220,10.187,149.553
C08073=1120.018,274.862,-73.785,-178.217,10.190,149.553
C08074=1120.014,275.110,-73.815,-178.214,10.193,149.553
C08075=1120.011,275.359,-73.845,-178.211,10.196,149.553
C08076=1120.006,275.607,-73.876,-178.207,10.198,149.553
C08077=1120.002,275.855,-73.905,-178.204,10.201,149.553
C08078=1119.998,276.103,-73.936,-178.201,10.204,149.553
C08079=1119.993,276.351,-73.966,-178.199,10.206,149.552
C08080=1119.989,276.599,-73.996,-178.195,10.209,149.552
C08081=1119.985,276.847,-74.025,-178.192,10.212,149.552
C08082=1119.981,277.096,-74.056,-178.189,10.214,149.552
C08083=1119.977,277.344,-74.086,-178.186,10.217,149.552
C08084=1119.973,277.592,-74.116,-178.183,10.219,149.552
C08085=1119.968,277.840,-74.146,-178.180,10.222,149.551
C08086=1119.964,278.088,-74.176,-178.177,10.225,149.551
C08087=1119.960,278.336,-74.206,-178.174,10.227,149.551
C08088=1119.956,278.585,-74.237,-178.171,10.230,149.551
C08089=1119.952,278.833,-74.267,-178.167,10.233,149.551
C08090=1119.947,279.081,-74.297,-178.164,10.236,149.551
C08091=1119.943,279.329,-74.327,-178.161,10.239,149.550
C08092=1119.939,279.577,-74.358,-178.158,10.241,149.550
C08093=1119.935,279.826,-74.388,-178.154,10.244,149.550
C08094=1119.932,280.039,-74.414,-178.151,10.246,149.550
C08095=1119.928,280.252,-74.440,-178.149,10.248,149.550
C08096=1119.925,280.464,-74.466,-178.146,10.251,149.550
C08097=1119.921,280.678,-74.493,-178.143,10.253,149.549
C08098=1119.917,280.890,-74.518,-178.141,10.256,149.549
C08099=1119.913,281.103,-74.545,-178.137,10.258,149.549
C08100=1119.910,281.316,-74.571,-178.135,10.260,149.549
C08101=1119.906,281.530,-74.597,-178.132,10.263,149.549
C08102=1119.902,281.778,-74.627,-178.129,10.265,149.548
C08103=1119.897,282.026,-74.658,-178.126,10.268,149.548
C08104=1119.894,282.274,-74.688,-178.123,10.270,149.548
C08105=1119.889,282.522,-74.719,-178.120,10.272,149.548
C08106=1119.886,282.770,-74.749,-178.117,10.275,149.548
C08107=1119.881,283.017,-74.780,-178.114,10.278,149.548
C08108=1119.877,283.266,-74.810,-178.111,10.280,149.548
C08109=1119.873,283.514,-74.840,-178.107,10.283,149.547
C08110=1119.868,283.762,-74.871,-178.104,10.285,149.547
C08111=1119.865,284.011,-74.902,-178.102,10.288,149.547
C08112=1119.860,284.259,-74.932,-178.098,10.291,149.547
C08113=1119.856,284.507,-74.963,-178.096,10.293,149.547
C08114=1119.852,284.754,-74.993,-178.093,10.295,149.546
C08115=1119.848,285.003,-75.024,-178.090,10.298,149.546
C08116=1119.843,285.251,-75.055,-178.086,10.300,149.546
C08117=1119.839,285.499,-75.085,-178.083,10.303,149.546
C08118=1119.835,285.747,-75.117,-178.080,10.306,149.546
C08119=1119.831,285.995,-75.147,-178.077,10.308,149.546
C08120=1119.827,286.243,-75.177,-178.074,10.311,149.545
C08121=1119.823,286.491,-75.209,-178.071,10.313,149.545
C08122=1119.818,286.739,-75.239,-178.068,10.315,149.545
C08123=1119.815,286.987,-75.271,-178.065,10.318,149.545
C08124=1119.811,287.235,-75.301,-178.062,10.321,149.545
C08125=1119.806,287.483,-75.332,-178.059,10.323,149.545
C08126=1119.802,287.732,-75.363,-178.056,10.326,149.544
C08127=1119.798,287.979,-75.393,-178.053,10.328,149.544
C08128=1119.794,288.227,-75.424,-178.050,10.331,149.544
C08129=1119.790,288.475,-75.456,-178.047,10.334,149.544
C08130=1119.785,288.723,-75.487,-178.043,10.336,149.544
C08131=1119.782,288.972,-75.517,-178.040,10.339,149.544
C08132=1119.777,289.220,-75.548,-178.038,10.340,149.543
C08133=1119.773,289.468,-75.579,-178.035,10.343,149.543
C08134=1119.769,289.716,-75.611,-178.032,10.346,149.543
C08135=1119.764,289.964,-75.641,-178.029,10.348,149.543
C08136=1119.761,290.212,-75.672,-178.026,10.351,149.543
C08137=1119.757,290.459,-75.704,-178.022,10.354,149.542
C08138=1119.753,290.708,-75.735,-178.019,10.356,149.542
C08139=1119.748,290.956,-75.765,-178.016,10.359,149.542
C08140=1119.744,291.204,-75.797,-178.013,10.362,149.542
C08141=1119.740,291.452,-75.828,-178.010,10.363,149.542
C08142=1119.736,291.701,-75.859,-178.007,10.366,149.542
C08143=1119.732,291.948,-75.890,-178.004,10.368,149.541
C08144=1119.728,292.196,-75.921,-178.001,10.371,149.541
C08145=1119.724,292.444,-75.952,-177.998,10.374,149.541
C08146=1119.719,292.692,-75.983,-177.995,10.376,149.541
C08147=1119.715,292.940,-76.015,-177.992,10.379,149.541
C08148=1119.711,293.188,-76.046,-177.989,10.382,149.540
C08149=1119.707,293.436,-76.077,-177.986,10.384,149.540
C08150=1119.703,293.649,-76.104,-177.983,10.386,149.540
C08151=1119.701,293.862,-76.131,-177.981,10.388,149.540
C08152=1119.697,294.075,-76.158,-177.978,10.391,149.540
C08153=1119.693,294.288,-76.184,-177.975,10.393,149.540
C08154=1119.689,294.500,-76.212,-177.973,10.394,149.539
C08155=1119.686,294.713,-76.239,-177.970,10.397,149.539
C08156=1119.682,294.927,-76.266,-177.967,10.399,149.539
C08157=1119.679,295.139,-76.292,-177.965,10.401,149.539
C08158=1119.675,295.387,-76.323,-177.962,10.404,149.539
C08159=1119.671,295.635,-76.355,-177.959,10.406,149.539
C08160=1119.667,295.883,-76.387,-177.956,10.409,149.539
C08161=1119.663,296.131,-76.417,-177.953,10.412,149.538
C08162=1119.658,296.379,-76.450,-177.949,10.414,149.538
C08163=1119.654,296.628,-76.481,-177.946,10.417,149.538
C08164=1119.650,296.875,-76.512,-177.943,10.419,149.538
C08165=1119.646,297.123,-76.544,-177.940,10.422,149.538
C08166=1119.642,297.371,-76.575,-177.937,10.424,149.537
C08167=1119.638,297.619,-76.607,-177.934,10.427,149.537
C08168=1119.633,297.866,-76.638,-177.931,10.429,149.537
C08169=1119.630,298.114,-76.670,-177.928,10.432,149.537
C08170=1119.626,298.363,-76.701,-177.925,10.434,149.537
C08171=1119.621,298.610,-76.733,-177.922,10.437,149.537
C08172=1119.617,298.859,-76.765,-177.919,10.439,149.536
C08173=1119.613,299.107,-76.797,-177.916,10.442,149.536
C08174=1119.609,299.355,-76.828,-177.912,10.444,149.536
C08175=1119.605,299.603,-76.860,-177.909,10.447,149.536
C08176=1119.601,299.850,-76.891,-177.906,10.450,149.536
C08177=1119.597,300.098,-76.923,-177.903,10.452,149.536
C08178=1119.593,300.347,-76.956,-177.900,10.454,149.535
C08179=1119.588,300.594,-76.987,-177.898,10.457,149.535
C08180=1119.585,300.842,-77.019,-177.894,10.459,149.535
C08181=1119.581,301.091,-77.050,-177.891,10.462,149.535
C08182=1119.576,301.338,-77.081,-177.888,10.464,149.535
C08183=1119.572,301.586,-77.114,-177.885,10.467,149.535
C08184=1119.568,301.834,-77.146,-177.882,10.470,149.534
C08185=1119.564,302.082,-77.177,-177.879,10.472,149.534
C08186=1119.560,302.330,-77.209,-177.875,10.475,149.534
C08187=1119.556,302.578,-77.241,-177.872,10.478,149.534
C08188=1119.551,302.825,-77.273,-177.869,10.480,149.534
C08189=1119.548,303.073,-77.305,-177.867,10.482,149.534
C08190=1119.543,303.322,-77.337,-177.863,10.484,149.533
C08191=1119.539,303.570,-77.369,-177.861,10.487,149.533
C08192=1119.535,303.817,-77.401,-177.857,10.490,149.533
C08193=1119.531,304.066,-77.433,-177.854,10.492,149.533
C08194=1119.527,304.314,-77.465,-177.851,10.495,149.533
C08195=1119.523,304.561,-77.496,-177.848,10.497,149.532
C08196=1119.519,304.809,-77.529,-177.845,10.500,149.532
C08197=1119.515,305.057,-77.561,-177.841,10.502,149.532
C08198=1119.511,305.305,-77.593,-177.838,10.505,149.532
C08199=1119.506,305.552,-77.625,-177.835,10.508,149.532
C08200=1119.502,305.800,-77.657,-177.833,10.510,149.532
C08201=1119.498,306.049,-77.690,-177.829,10.512,149.531
C08202=1119.494,306.297,-77.721,-177.827,10.515,149.531
C08203=1119.491,306.544,-77.754,-177.823,10.517,149.531
C08204=1119.486,306.792,-77.786,-177.820,10.520,149.531
C08205=1119.482,307.040,-77.818,-177.817,10.522,149.531
C08206=1119.478,307.253,-77.846,-177.815,10.524,149.530
C08207=1119.475,307.465,-77.874,-177.811,10.527,149.530
C08208=1119.472,307.678,-77.902,-177.809,10.529,149.530
C08209=1119.468,307.891,-77.929,-177.807,10.531,149.530
C08210=1119.465,308.104,-77.956,-177.803,10.533,149.530
C08211=1119.461,308.316,-77.985,-177.801,10.535,149.530
C08212=1119.457,308.529,-78.012,-177.798,10.538,149.530
C08213=1119.454,308.742,-78.040,-177.795,10.540,149.529
C08214=1119.450,308.990,-78.072,-177.793,10.542,149.529
C08215=1119.446,309.238,-78.105,-177.789,10.545,149.529
C08216=1119.442,309.486,-78.137,-177.786,10.548,149.529
C08217=1119.438,309.733,-78.169,-177.783,10.550,149.529
C08218=1119.433,309.981,-78.202,-177.781,10.552,149.529
C08219=1119.430,310.229,-78.234,-177.777,10.555,149.528
C08220=1119.426,310.477,-78.267,-177.774,10.557,149.528
C08221=1119.422,310.725,-78.299,-177.771,10.560,149.528
C08222=1119.418,310.973,-78.332,-177.768,10.562,149.528
C08223=1119.413,311.221,-78.364,-177.765,10.565,149.528
C08224=1119.410,311.468,-78.397,-177.761,10.567,149.527
C08225=1119.405,311.716,-78.429,-177.759,10.570,149.527
C08226=1119.401,311.964,-78.461,-177.755,10.573,149.527
C08227=1119.397,312.212,-78.494,-177.752,10.575,149.527
C08228=1119.393,312.460,-78.527,-177.749,10.578,149.527
C08229=1119.389,312.708,-78.559,-177.746,10.580,149.526
C08230=1119.385,312.955,-78.592,-177.743,10.582,149.526
C08231=1119.381,313.203,-78.624,-177.740,10.585,149.526
C08232=1119.377,313.451,-78.657,-177.737,10.587,149.526
C08233=1119.373,313.699,-78.690,-177.734,10.590,149.526
C08234=1119.369,313.947,-78.722,-177.730,10.592,149.525
C08235=1119.365,314.195,-78.755,-177.728,10.595,149.525
C08236=1119.361,314.442,-78.788,-177.724,10.598,149.525
C08237=1119.357,314.690,-78.820,-177.721,10.600,149.525
C08238=1119.353,314.938,-78.853,-177.718,10.603,149.525
C08239=1119.349,315.186,-78.886,-177.715,10.605,149.525
C08240=1119.345,315.434,-78.919,-177.712,10.608,149.525
C08241=1119.341,315.682,-78.951,-177.708,10.610,149.524
C08242=1119.337,315.929,-78.985,-177.706,10.612,149.524
C08243=1119.333,316.177,-79.018,-177.703,10.615,149.524
C08244=1119.328,316.425,-79.050,-177.699,10.617,149.524
C08245=1119.325,316.673,-79.083,-177.696,10.620,149.524
C08246=1119.321,316.921,-79.116,-177.693,10.623,149.523
C08247=1119.317,317.168,-79.149,-177.690,10.625,149.523
C08248=1119.313,317.416,-79.182,-177.687,10.628,149.523
C08249=1119.309,317.664,-79.214,-177.684,10.630,149.523
C08250=1119.305,317.912,-79.247,-177.681,10.633,149.523
C08251=1119.301,318.160,-79.280,-177.677,10.635,149.522
C08252=1119.297,318.407,-79.313,-177.674,10.638,149.522
C08253=1119.292,318.655,-79.347,-177.671,10.641,149.522
C08254=1119.288,318.903,-79.380,-177.668,10.643,149.522
C08255=1119.285,319.150,-79.412,-177.665,10.645,149.522
C08256=1119.281,319.398,-79.446,-177.662,10.648,149.522
C08257=1119.277,319.646,-79.479,-177.659,10.650,149.521
C08258=1119.272,319.893,-79.512,-177.656,10.653,149.521
C08259=1119.268,320.141,-79.545,-177.653,10.655,149.521
C08260=1119.265,320.390,-79.579,-177.650,10.658,149.521
C08261=1119.261,320.637,-79.612,-177.646,10.660,149.521
C08262=1119.257,320.849,-79.640,-177.644,10.662,149.520
C08263=1119.253,321.063,-79.668,-177.641,10.665,149.520
C08264=1119.251,321.275,-79.696,-177.638,10.667,149.520
C08265=1119.246,321.487,-79.725,-177.636,10.668,149.520
C08266=1119.243,321.700,-79.753,-177.633,10.671,149.520
C08267=1119.240,321.913,-79.782,-177.630,10.673,149.520
C08268=1119.237,322.126,-79.811,-177.628,10.675,149.519
C08269=1119.233,322.338,-79.839,-177.625,10.678,149.519
C08270=1119.230,322.586,-79.872,-177.622,10.680,149.519
C08271=1119.226,322.834,-79.905,-177.618,10.683,149.519
C08272=1119.222,323.081,-79.939,-177.615,10.685,149.519
C08273=1119.218,323.329,-79.972,-177.612,10.688,149.519
C08274=1119.214,323.576,-80.005,-177.609,10.689,149.518
C08275=1119.209,323.824,-80.039,-177.606,10.692,149.518
C08276=1119.206,324.072,-80.072,-177.603,10.695,149.518
C08277=1119.202,324.320,-80.106,-177.600,10.697,149.518
C08278=1119.198,324.567,-80.139,-177.597,10.700,149.518
C08279=1119.194,324.815,-80.172,-177.593,10.702,149.517
C08280=1119.190,325.063,-80.205,-177.590,10.705,149.517
C08281=1119.185,325.310,-80.240,-177.587,10.708,149.517
C08282=1119.181,325.559,-80.273,-177.584,10.710,149.517
C08283=1119.177,325.806,-80.307,-177.581,10.712,149.517
C08284=1119.173,326.054,-80.340,-177.578,10.715,149.517
C08285=1119.169,326.301,-80.374,-177.574,10.718,149.516
C08286=1119.165,326.549,-80.407,-177.571,10.720,149.516
C08287=1119.162,326.797,-80.441,-177.569,10.722,149.516
C08288=1119.158,327.044,-80.474,-177.565,10.725,149.516
C08289=1119.154,327.292,-80.507,-177.562,10.727,149.516
C08290=1119.149,327.540,-80.542,-177.559,10.730,149.515
C08291=1119.146,327.788,-80.575,-177.556,10.732,149.515
C08292=1119.142,328.035,-80.609,-177.552,10.735,149.515
C08293=1119.138,328.283,-80.642,-177.550,10.738,149.515
C08294=1119.134,328.531,-80.675,-177.546,10.740,149.515
C08295=1119.130,328.779,-80.710,-177.543,10.742,149.514
C08296=1119.125,329.026,-80.743,-177.540,10.745,149.514
C08297=1119.122,329.273,-80.777,-177.537,10.748,149.514
C08298=1119.118,329.522,-80.811,-177.533,10.750,149.514
C08299=1119.114,329.769,-80.845,-177.530,10.753,149.514
C08300=1119.110,330.016,-80.879,-177.528,10.755,149.514
C08301=1119.105,330.264,-80.912,-177.524,10.757,149.513
C08302=1119.102,330.512,-80.947,-177.521,10.759,149.513
C08303=1119.098,330.760,-80.980,-177.518,10.762,149.513
C08304=1119.094,331.007,-81.014,-177.515,10.765,149.513
C08305=1119.090,331.256,-81.048,-177.512,10.767,149.513
C08306=1119.086,331.503,-81.082,-177.508,10.770,149.512
C08307=1119.082,331.750,-81.116,-177.505,10.772,149.512
C08308=1119.078,331.999,-81.150,-177.502,10.775,149.512
C08309=1119.074,332.246,-81.183,-177.499,10.777,149.512
C08310=1119.070,332.493,-81.218,-177.496,10.780,149.512
C08311=1119.066,332.741,-81.252,-177.492,10.782,149.511
C08312=1119.062,332.989,-81.285,-177.489,10.785,149.511
C08313=1119.058,333.237,-81.320,-177.486,10.787,149.511
C08314=1119.055,333.484,-81.354,-177.484,10.789,149.511
C08315=1119.050,333.732,-81.387,-177.480,10.792,149.511
C08316=1119.046,333.980,-81.422,-177.477,10.794,149.510
C08317=1119.043,334.227,-81.456,-177.474,10.797,149.510
C08318=1119.039,334.439,-81.485,-177.471,10.800,149.510
C08319=1119.036,334.652,-81.514,-177.468,10.802,149.510
C08320=1119.033,334.864,-81.544,-177.466,10.803,149.510
C08321=1119.029,335.077,-81.573,-177.463,10.806,149.510
C08322=1119.026,335.289,-81.602,-177.460,10.808,149.509
C08323=1119.023,335.502,-81.632,-177.458,10.810,149.509
C08324=1119.019,335.714,-81.661,-177.454,10.812,149.509
C08325=1119.015,335.926,-81.690,-177.452,10.814,149.509
C08326=1119.011,336.174,-81.725,-177.449,10.817,149.509
C08327=1119.008,336.421,-81.759,-177.446,10.819,149.509
C08328=1119.004,336.669,-81.794,-177.442,10.821,149.508
C08329=1119.000,336.916,-81.828,-177.439,10.824,149.508
C08330=1118.996,337.165,-81.862,-177.436,10.827,149.508
C08331=1118.992,337.412,-81.896,-177.433,10.829,149.508
C08332=1118.988,337.660,-81.931,-177.429,10.832,149.508
C08333=1118.984,337.907,-81.965,-177.426,10.834,149.507
C08334=1118.980,338.155,-82.000,-177.423,10.837,149.507
C08335=1118.976,338.402,-82.034,-177.420,10.839,149.507
C08336=1118.972,338.650,-82.069,-177.417,10.841,149.507
C08337=1118.969,338.897,-82.102,-177.414,10.843,149.507
C08338=1118.964,339.145,-82.137,-177.411,10.846,149.506
C08339=1118.961,339.393,-82.171,-177.408,10.849,149.506
C08340=1118.956,339.640,-82.206,-177.404,10.851,149.506
C08341=1118.952,339.888,-82.240,-177.401,10.854,149.506
C08342=1118.948,340.135,-82.274,-177.398,10.856,149.506
C08343=1118.944,340.383,-82.309,-177.395,10.859,149.505
C08344=1118.940,340.630,-82.344,-177.391,10.861,149.505
C08345=1118.937,340.878,-82.379,-177.388,10.864,149.505
C08346=1118.933,341.126,-82.413,-177.385,10.866,149.505
C08347=1118.928,341.374,-82.448,-177.382,10.869,149.505
C08348=1118.925,341.621,-82.482,-177.379,10.871,149.504
C08349=1118.921,341.868,-82.517,-177.376,10.873,149.504
C08350=1118.917,342.116,-82.552,-177.372,10.876,149.504
C08351=1118.913,342.363,-82.586,-177.369,10.878,149.504
C08352=1118.909,342.611,-82.621,-177.366,10.881,149.504
C08353=1118.905,342.858,-82.656,-177.363,10.883,149.503
C08354=1118.902,343.106,-82.690,-177.360,10.886,149.503
C08355=1118.897,343.353,-82.725,-177.356,10.888,149.503
C08356=1118.893,343.601,-82.760,-177.353,10.891,149.503
C08357=1118.889,343.849,-82.795,-177.350,10.893,149.503
C08358=1118.886,344.096,-82.829,-177.347,10.896,149.503
C08359=1118.882,344.344,-82.864,-177.343,10.898,149.502
C08360=1118.877,344.591,-82.899,-177.340,10.901,149.502
C08361=1118.874,344.839,-82.934,-177.337,10.903,149.502
C08362=1118.870,345.086,-82.969,-177.334,10.905,149.502
C08363=1118.866,345.334,-83.003,-177.331,10.908,149.502
C08364=1118.862,345.581,-83.039,-177.328,10.910,149.501
C08365=1118.858,345.830,-83.074,-177.325,10.913,149.501
C08366=1118.854,346.076,-83.109,-177.321,10.915,149.501
C08367=1118.851,346.324,-83.143,-177.318,10.918,149.501
C08368=1118.847,346.572,-83.179,-177.315,10.920,149.500
C08369=1118.843,346.819,-83.213,-177.312,10.923,149.500
C08370=1118.839,347.067,-83.249,-177.308,10.925,149.500
C08371=1118.834,347.314,-83.283,-177.305,10.928,149.500
C08372=1118.831,347.561,-83.319,-177.302,10.930,149.500
C08373=1118.827,347.810,-83.353,-177.299,10.933,149.499
C08374=1118.824,348.021,-83.384,-177.296,10.935,149.499
C08375=1118.821,348.233,-83.413,-177.294,10.936,149.499
C08376=1118.817,348.446,-83.443,-177.290,10.939,149.499
C08377=1118.814,348.658,-83.474,-177.288,10.941,149.499
C08378=1118.810,348.871,-83.504,-177.285,10.943,149.499
C08379=1118.807,349.083,-83.534,-177.282,10.945,149.498
C08380=1118.803,349.295,-83.565,-177.280,10.947,149.498
C08381=1118.800,349.507,-83.594,-177.276,10.949,149.498
C08382=1118.797,349.755,-83.630,-177.273,10.952,149.498
C08383=1118.793,350.003,-83.665,-177.270,10.954,149.498
C08384=1118.788,350.250,-83.700,-177.266,10.957,149.497
C08385=1118.785,350.497,-83.736,-177.263,10.959,149.497
C08386=1118.781,350.745,-83.771,-177.259,10.963,149.497
C08387=1118.777,350.993,-83.806,-177.256,10.965,149.497
C08388=1118.773,351.240,-83.841,-177.253,10.967,149.496
C08389=1118.769,351.487,-83.877,-177.249,10.970,149.496
C08390=1118.765,351.735,-83.912,-177.246,10.972,149.496
C08391=1118.762,351.982,-83.948,-177.242,10.974,149.496
C08392=1118.757,352.230,-83.982,-177.239,10.977,149.495
C08393=1118.754,352.477,-84.018,-177.235,10.980,149.495
C08394=1118.750,352.725,-84.053,-177.232,10.983,149.495
C08395=1118.746,352.972,-84.089,-177.228,10.985,149.495
C08396=1118.743,353.220,-84.124,-177.225,10.988,149.494
C08397=1118.738,353.466,-84.160,-177.222,10.990,149.494
C08398=1118.735,353.714,-84.195,-177.218,10.992,149.494
C08399=1118.731,353.961,-84.231,-177.215,10.995,149.494
C08400=1118.727,354.209,-84.266,-177.211,10.997,149.493
C08401=1118.723,354.457,-84.302,-177.208,11.000,149.493
C08402=1118.719,354.704,-84.338,-177.204,11.003,149.493
C08403=1118.715,354.951,-84.373,-177.201,11.005,149.493
C08404=1118.711,355.199,-84.409,-177.197,11.007,149.492
C08405=1118.708,355.446,-84.444,-177.194,11.010,149.492
C08406=1118.704,355.694,-84.480,-177.191,11.012,149.492
C08407=1118.700,355.941,-84.515,-177.187,11.015,149.492
C08408=1118.696,356.189,-84.551,-177.184,11.017,149.491
C08409=1118.692,356.436,-84.587,-177.180,11.019,149.491
C08410=1118.689,356.684,-84.623,-177.177,11.022,149.491
C08411=1118.684,356.931,-84.658,-177.174,11.024,149.491
C08412=1118.681,357.178,-84.694,-177.170,11.027,149.490
C08413=1118.677,357.425,-84.730,-177.167,11.029,149.490
C08414=1118.673,357.673,-84.766,-177.163,11.031,149.490
C08415=1118.669,357.920,-84.801,-177.160,11.034,149.490
C08416=1118.666,358.168,-84.837,-177.157,11.036,149.489
C08417=1118.662,358.415,-84.873,-177.153,11.039,149.489
C08418=1118.658,358.663,-84.909,-177.150,11.041,149.489
C08419=1118.654,358.910,-84.945,-177.146,11.043,149.489
C08420=1118.651,359.158,-84.980,-177.143,11.046,149.488
C08421=1118.646,359.405,-85.017,-177.139,11.049,149.488
C08422=1118.643,359.652,-85.053,-177.136,11.052,149.488
C08423=1118.639,359.900,-85.088,-177.132,11.054,149.487
C08424=1118.636,360.147,-85.125,-177.129,11.056,149.487
C08425=1118.631,360.394,-85.161,-177.125,11.059,149.487
C08426=1118.628,360.642,-85.196,-177.122,11.061,149.487
C08427=1118.624,360.889,-85.232,-177.118,11.063,149.486
C08428=1118.620,361.137,-85.269,-177.115,11.066,149.486
C08429=1118.617,361.384,-85.305,-177.113,11.067,149.486
C08430=1118.613,361.595,-85.336,-177.109,11.070,149.486
C08431=1118.609,361.807,-85.367,-177.107,11.072,149.486
C08432=1118.607,362.020,-85.397,-177.103,11.074,149.485
C08433=1118.603,362.232,-85.428,-177.101,11.076,149.485
C08434=1118.600,362.444,-85.460,-177.098,11.079,149.485
C08435=1118.597,362.656,-85.490,-177.095,11.080,149.485
C08436=1118.594,362.869,-85.522,-177.092,11.082,149.484
C08437=1118.590,363.081,-85.553,-177.089,11.084,149.484
C08438=1118.586,363.328,-85.588,-177.086,11.087,149.484
C08439=1118.583,363.575,-85.624,-177.082,11.089,149.484
C08440=1118.579,363.822,-85.661,-177.079,11.092,149.483
C08441=1118.575,364.070,-85.697,-177.075,11.094,149.483
C08442=1118.571,364.317,-85.734,-177.072,11.096,149.483
C08443=1118.567,364.565,-85.769,-177.069,11.099,149.483
C08444=1118.563,364.812,-85.806,-177.066,11.100,149.482
C08445=1118.560,365.059,-85.842,-177.062,11.103,149.482
C08446=1118.556,365.307,-85.879,-177.059,11.105,149.482
C08447=1118.553,365.554,-85.915,-177.056,11.108,149.482
C08448=1118.549,365.801,-85.952,-177.052,11.110,149.482
C08449=1118.545,366.049,-85.988,-177.049,11.113,149.481
C08450=1118.541,366.296,-86.024,-177.045,11.115,149.481
C08451=1118.538,366.543,-86.061,-177.042,11.117,149.481
C08452=1118.533,366.791,-86.097,-177.039,11.120,149.481
C08453=1118.529,367.038,-86.134,-177.036,11.122,149.480
C08454=1118.526,367.285,-86.170,-177.032,11.125,149.480
C08455=1118.522,367.532,-86.207,-177.029,11.127,149.480
C08456=1118.519,367.780,-86.243,-177.026,11.130,149.480
C08457=1118.515,368.027,-86.280,-177.022,11.132,149.479
C08458=1118.510,368.275,-86.316,-177.019,11.134,149.479
C08459=1118.507,368.521,-86.353,-177.016,11.136,149.479
C08460=1118.503,368.769,-86.390,-177.013,11.138,149.479
C08461=1118.500,369.015,-86.426,-177.009,11.141,149.478
C08462=1118.496,369.264,-86.462,-177.006,11.143,149.478
C08463=1118.492,369.511,-86.499,-177.003,11.146,149.478
C08464=1118.488,369.758,-86.535,-177.000,11.148,149.478
C08465=1118.484,370.005,-86.572,-176.996,11.151,149.478
C08466=1118.480,370.252,-86.609,-176.993,11.153,149.477
C08467=1118.477,370.499,-86.645,-176.990,11.156,149.477
C08468=1118.473,370.747,-86.683,-176.986,11.158,149.477
C08469=1118.469,370.994,-86.720,-176.983,11.160,149.477
C08470=1118.465,371.242,-86.756,-176.980,11.162,149.476
C08471=1118.462,371.488,-86.793,-176.977,11.165,149.476
C08472=1118.458,371.736,-86.830,-176.973,11.167,149.476
C08473=1118.454,371.984,-86.867,-176.970,11.170,149.476
C08474=1118.451,372.230,-86.903,-176.967,11.172,149.475
C08475=1118.447,372.478,-86.940,-176.963,11.174,149.475
C08476=1118.443,372.725,-86.977,-176.960,11.177,149.475
C08477=1118.439,372.973,-87.014,-176.957,11.179,149.475
C08478=1118.435,373.220,-87.051,-176.954,11.182,149.475
C08479=1118.432,373.466,-87.088,-176.950,11.184,149.474
C08480=1118.429,373.714,-87.125,-176.948,11.186,149.474
C08481=1118.424,373.961,-87.162,-176.945,11.189,149.474
C08482=1118.420,374.208,-87.199,-176.941,11.191,149.474
C08483=1118.416,374.456,-87.236,-176.938,11.194,149.474
C08484=1118.413,374.703,-87.272,-176.935,11.196,149.474
C08485=1118.410,374.950,-87.310,-176.932,11.199,149.473
C08486=1118.406,375.163,-87.342,-176.929,11.201,149.473
C08487=1118.403,375.374,-87.373,-176.926,11.203,149.473
C08488=1118.400,375.586,-87.405,-176.923,11.205,149.473
C08489=1118.396,375.797,-87.437,-176.921,11.207,149.473
C08490=1118.393,376.010,-87.468,-176.918,11.210,149.473
C08491=1118.390,376.222,-87.501,-176.915,11.211,149.472
C08492=1118.387,376.434,-87.532,-176.913,11.213,149.472
C08493=1118.384,376.646,-87.564,-176.909,11.216,149.472
C08494=1118.380,376.893,-87.601,-176.906,11.218,149.472
C08495=1118.376,377.141,-87.638,-176.904,11.220,149.472
C08496=1118.373,377.387,-87.676,-176.901,11.223,149.472
C08497=1118.368,377.635,-87.713,-176.897,11.225,149.471
C08498=1118.365,377.882,-87.750,-176.894,11.228,149.471
C08499=1118.361,378.129,-87.788,-176.891,11.231,149.471
C08500=1118.357,378.376,-87.825,-176.888,11.233,149.471
C08501=1118.354,378.623,-87.862,-176.885,11.236,149.471
C08502=1118.350,378.871,-87.899,-176.881,11.238,149.471
C08503=1118.346,379.117,-87.937,-176.878,11.241,149.471
C08504=1118.342,379.365,-87.974,-176.875,11.243,149.470
C08505=1118.338,379.612,-88.011,-176.872,11.245,149.470
C08506=1118.335,379.860,-88.049,-176.869,11.248,149.470
C08507=1118.331,380.107,-88.086,-176.866,11.250,149.470
C08508=1118.327,380.353,-88.123,-176.863,11.253,149.470
C08509=1118.324,380.601,-88.161,-176.860,11.256,149.470
C08510=1118.320,380.848,-88.198,-176.857,11.258,149.470
C08511=1118.317,381.095,-88.236,-176.854,11.261,149.470
C08512=1118.313,381.342,-88.273,-176.851,11.263,149.469
C08513=1118.309,381.589,-88.311,-176.848,11.266,149.469
C08514=1118.305,381.837,-88.348,-176.844,11.269,149.469
C08515=1118.302,382.083,-88.385,-176.841,11.272,149.469
C08516=1118.298,382.331,-88.423,-176.839,11.273,149.469
C08517=1118.294,382.578,-88.460,-176.836,11.276,149.469
C08518=1118.290,382.825,-88.499,-176.833,11.279,149.469
C08519=1118.287,383.072,-88.536,-176.830,11.281,149.469
C08520=1118.283,383.320,-88.573,-176.827,11.284,149.469
C08521=1118.279,383.566,-88.611,-176.823,11.287,149.469
C08522=1118.276,383.814,-88.649,-176.822,11.289,149.469
C08523=1118.272,384.060,-88.687,-176.819,11.291,149.469
C08524=1118.269,384.308,-88.724,-176.817,11.293,149.469
C08525=1118.264,384.555,-88.762,-176.815,11.295,149.469
C08526=1118.261,384.802,-88.800,-176.813,11.297,149.469
C08527=1118.257,385.049,-88.837,-176.811,11.299,149.469
C08528=1118.253,385.296,-88.874,-176.809,11.302,149.469
C08529=1118.250,385.543,-88.912,-176.806,11.305,149.469
C08530=1118.247,385.791,-88.950,-176.804,11.307,149.469
C08531=1118.242,386.037,-88.988,-176.802,11.309,149.469
C08532=1118.239,386.285,-89.026,-176.800,11.311,149.469
C08533=1118.235,386.532,-89.063,-176.798,11.314,149.469
C08534=1118.232,386.779,-89.101,-176.795,11.317,149.469
C08535=1118.227,387.026,-89.139,-176.793,11.319,149.469
C08536=1118.224,387.273,-89.177,-176.791,11.321,149.469
C08537=1118.220,387.520,-89.215,-176.789,11.324,149.469
C08538=1118.217,387.767,-89.253,-176.787,11.327,149.470
C08539=1118.213,388.014,-89.290,-176.785,11.329,149.470
C08540=1118.210,388.261,-89.329,-176.783,11.331,149.470
C08541=1118.206,388.508,-89.366,-176.781,11.334,149.470
C08542=1118.202,388.720,-89.399,-176.779,11.336,149.470
C08543=1118.200,388.932,-89.431,-176.777,11.338,149.470
C08544=1118.196,389.144,-89.464,-176.775,11.341,149.470
C08545=1118.194,389.356,-89.496,-176.773,11.343,149.470
C08546=1118.190,389.568,-89.529,-176.772,11.346,149.471
C08547=1118.187,389.779,-89.561,-176.770,11.348,149.471
C08548=1118.184,389.991,-89.594,-176.769,11.350,149.471
C08549=1118.181,390.203,-89.626,-176.767,11.352,149.471
C08550=1118.177,390.450,-89.665,-176.764,11.355,149.471
C08551=1118.174,390.697,-89.703,-176.763,11.358,149.472
C08552=1118.170,390.944,-89.741,-176.761,11.360,149.472
C08553=1118.166,391.191,-89.779,-176.759,11.364,149.472
C08554=1118.163,391.438,-89.817,-176.757,11.366,149.472
C08555=1118.159,391.686,-89.855,-176.755,11.369,149.473
C08556=1118.155,391.932,-89.893,-176.753,11.372,149.473
C08557=1118.152,392.180,-89.931,-176.751,11.375,149.473
C08558=1118.149,392.427,-89.969,-176.749,11.378,149.473
C08559=1118.144,392.674,-90.007,-176.747,11.381,149.474
C08560=1118.141,392.921,-90.045,-176.746,11.384,149.474
C08561=1118.137,393.167,-90.084,-176.743,11.387,149.474
C08562=1118.133,393.415,-90.122,-176.742,11.390,149.474
C08563=1118.130,393.662,-90.160,-176.739,11.393,149.475
C08564=1118.126,393.909,-90.198,-176.738,11.396,149.475
C08565=1118.123,394.156,-90.236,-176.736,11.399,149.475
C08566=1118.119,394.403,-90.275,-176.734,11.402,149.476
C08567=1118.115,394.650,-90.312,-176.732,11.405,149.476
C08568=1118.111,394.897,-90.351,-176.731,11.408,149.476
C08569=1118.108,395.145,-90.389,-176.729,11.412,149.477
C08570=1118.103,395.391,-90.427,-176.727,11.415,149.477
C08571=1118.101,395.638,-90.466,-176.726,11.418,149.478
C08572=1118.097,395.885,-90.504,-176.723,11.422,149.478
C08573=1118.093,396.132,-90.542,-176.721,11.425,149.478
C08574=1118.090,396.379,-90.581,-176.720,11.428,149.479
C08575=1118.086,396.626,-90.619,-176.718,11.431,149.479
C08576=1118.082,396.873,-90.657,-176.716,11.435,149.480
C08577=1118.078,397.121,-90.695,-176.715,11.438,149.480
C08578=1118.075,397.367,-90.734,-176.713,11.442,149.481
C08579=1118.071,397.614,-90.772,-176.711,11.445,149.481
C08580=1118.068,397.861,-90.811,-176.709,11.449,149.482
C08581=1118.064,398.108,-90.849,-176.708,11.452,149.482
C08582=1118.060,398.356,-90.888,-176.707,11.456,149.483
C08583=1118.057,398.602,-90.926,-176.705,11.460,149.483
C08584=1118.053,398.849,-90.965,-176.703,11.463,149.484
C08585=1118.050,399.096,-91.003,-176.701,11.467,149.484
C08586=1118.046,399.344,-91.042,-176.700,11.470,149.485
C08587=1118.042,399.590,-91.079,-176.698,11.474,149.485
C08588=1118.039,399.837,-91.119,-176.697,11.478,149.486
C08589=1118.035,400.084,-91.156,-176.695,11.482,149.487
C08590=1118.032,400.331,-91.196,-176.693,11.485,149.487
C08591=1118.027,400.578,-91.234,-176.692,11.489,149.488
C08592=1118.024,400.825,-91.273,-176.690,11.493,149.488
C08593=1118.020,401.073,-91.311,-176.689,11.497,149.489
C08594=1118.018,401.319,-91.350,-176.687,11.501,149.490
C08595=1118.013,401.566,-91.388,-176.686,11.505,149.490
C08596=1118.009,401.813,-91.427,-176.684,11.509,149.491
C08597=1118.006,402.060,-91.465,-176.683,11.513,149.492
C08598=1118.003,402.272,-91.498,-176.681,11.516,149.492
C08599=1118.000,402.484,-91.532,-176.680,11.520,149.493
C08600=1117.997,402.695,-91.565,-176.679,11.523,149.493
C08601=1117.994,402.907,-91.598,-176.678,11.526,149.494
C08602=1117.990,403.119,-91.632,-176.677,11.530,149.495
C08603=1117.988,403.330,-91.664,-176.676,11.533,149.495
C08604=1117.985,403.542,-91.698,-176.674,11.537,149.496
C08605=1117.982,403.754,-91.731,-176.673,11.540,149.496
C08606=1117.978,404.001,-91.770,-176.671,11.545,149.497
C08607=1117.974,404.248,-91.809,-176.670,11.550,149.498
C08608=1117.971,404.494,-91.847,-176.669,11.554,149.499
C08609=1117.967,404.741,-91.886,-176.668,11.558,149.500
C08610=1117.963,404.989,-91.925,-176.666,11.562,149.500
C08611=1117.960,405.235,-91.963,-176.665,11.567,149.501
C08612=1117.957,405.482,-92.003,-176.663,11.571,149.502
C08613=1117.953,405.729,-92.042,-176.662,11.576,149.503
C08614=1117.949,405.976,-92.080,-176.661,11.580,149.504
C08615=1117.946,406.223,-92.119,-176.660,11.584,149.505
C08616=1117.942,406.470,-92.158,-176.658,11.589,149.505
C08617=1117.938,406.717,-92.197,-176.657,11.594,149.506
C08618=1117.935,406.963,-92.236,-176.656,11.598,149.507
C08619=1117.931,407.211,-92.274,-176.655,11.604,149.508
C08620=1117.928,407.458,-92.314,-176.654,11.608,149.509
C08621=1117.924,407.705,-92.353,-176.653,11.612,149.510
C08622=1117.921,407.952,-92.392,-176.651,11.618,149.511
C08623=1117.917,408.198,-92.430,-176.650,11.622,149.512
C08624=1117.914,408.445,-92.470,-176.649,11.627,149.513
C08625=1117.910,408.692,-92.509,-176.648,11.632,149.514
C08626=1117.906,408.939,-92.548,-176.647,11.636,149.515
C08627=1117.902,409.186,-92.587,-176.646,11.642,149.516
C08628=1117.899,409.433,-92.625,-176.645,11.646,149.517
C08629=1117.896,409.680,-92.665,-176.643,11.652,149.518
C08630=1117.892,409.927,-92.704,-176.642,11.656,149.519
C08631=1117.889,410.174,-92.743,-176.641,11.662,149.520
C08632=1117.885,410.421,-92.782,-176.640,11.666,149.521
C08633=1117.881,410.668,-92.822,-176.639,11.672,149.522
C08634=1117.878,410.915,-92.861,-176.639,11.676,149.523
C08635=1117.874,411.162,-92.900,-176.637,11.682,149.524
C08636=1117.871,411.408,-92.939,-176.636,11.688,149.526
C08637=1117.868,411.655,-92.978,-176.636,11.692,149.527
C08638=1117.863,411.902,-93.017,-176.634,11.698,149.528
C08639=1117.860,412.149,-93.056,-176.633,11.703,149.529
C08640=1117.856,412.395,-93.095,-176.633,11.708,149.530
C08641=1117.853,412.642,-93.135,-176.631,11.714,149.531
C08642=1117.849,412.889,-93.175,-176.631,11.720,149.533
C08643=1117.846,413.136,-93.214,-176.630,11.724,149.534
C08644=1117.842,413.383,-93.253,-176.629,11.730,149.535
C08645=1117.838,413.630,-93.292,-176.628,11.736,149.536
C08646=1117.836,413.877,-93.331,-176.627,11.742,149.537
C08647=1117.833,414.124,-93.371,-176.626,11.748,149.539
C08648=1117.831,414.370,-93.410,-176.626,11.753,149.540
C08649=1117.829,414.618,-93.449,-176.625,11.758,149.541
C08650=1117.828,414.865,-93.488,-176.624,11.764,149.543
C08651=1117.828,415.112,-93.527,-176.623,11.770,149.544
C08652=1117.829,415.359,-93.566,-176.623,11.776,149.545
C08653=1117.829,415.605,-93.605,-176.622,11.782,149.547
C08654=1117.829,415.817,-93.638,-176.622,11.787,149.548
C08655=1117.831,416.028,-93.672,-176.621,11.792,149.549
C08656=1117.833,416.239,-93.704,-176.621,11.797,149.550
C08657=1117.835,416.451,-93.737,-176.621,11.802,149.552
C08658=1117.838,416.663,-93.771,-176.620,11.806,149.553
C08659=1117.840,416.874,-93.803,-176.619,11.812,149.554
C08660=1117.843,417.085,-93.836,-176.619,11.817,149.555
C08661=1117.848,417.297,-93.869,-176.618,11.822,149.556
C08662=1117.429,417.297,-93.932,-176.611,11.827,149.556
C08663=1117.424,417.085,-93.899,-176.612,11.822,149.555
C08664=1117.421,416.874,-93.866,-176.612,11.817,149.553
C08665=1117.419,416.662,-93.833,-176.613,11.811,149.552
C08666=1117.416,416.451,-93.800,-176.613,11.806,149.551
C08667=1117.414,416.239,-93.767,-176.613,11.801,149.550
C08668=1117.412,416.027,-93.734,-176.614,11.796,149.548
C08669=1117.411,415.817,-93.700,-176.614,11.791,149.547
C08670=1117.410,415.605,-93.668,-176.615,11.786,149.546
C08671=1117.409,415.358,-93.629,-176.616,11.780,149.545
C08672=1117.409,415.111,-93.590,-176.617,11.774,149.543
C08673=1117.409,414.864,-93.551,-176.617,11.769,149.542
C08674=1117.410,414.618,-93.512,-176.618,11.763,149.541
C08675=1117.412,414.370,-93.473,-176.619,11.757,149.539
C08676=1117.414,414.124,-93.433,-176.620,11.751,149.538
C08677=1117.417,413.876,-93.394,-176.621,11.746,149.537
C08678=1117.419,413.630,-93.355,-176.622,11.740,149.536
C08679=1117.423,413.383,-93.315,-176.623,11.734,149.534
C08680=1117.426,413.136,-93.276,-176.623,11.729,149.533
C08681=1117.430,412.889,-93.237,-176.624,11.723,149.532
C08682=1117.434,412.642,-93.197,-176.625,11.718,149.531
C08683=1117.437,412.395,-93.158,-176.626,11.712,149.529
C08684=1117.441,412.149,-93.119,-176.627,11.707,149.528
C08685=1117.444,411.902,-93.080,-176.628,11.702,149.527
C08686=1117.448,411.655,-93.040,-176.629,11.696,149.526
C08687=1117.451,411.408,-93.000,-176.630,11.691,149.525
C08688=1117.455,411.161,-92.961,-176.631,11.686,149.524
C08689=1117.459,410.914,-92.922,-176.632,11.680,149.523
C08690=1117.462,410.668,-92.883,-176.633,11.675,149.521
C08691=1117.465,410.421,-92.844,-176.634,11.670,149.521
C08692=1117.469,410.174,-92.805,-176.636,11.665,149.519
C08693=1117.472,409.927,-92.766,-176.637,11.660,149.518
C08694=1117.476,409.680,-92.726,-176.638,11.655,149.517
C08695=1117.480,409.433,-92.687,-176.639,11.650,149.516
C08696=1117.483,409.186,-92.648,-176.640,11.645,149.515
C08697=1117.486,408.939,-92.610,-176.641,11.640,149.514
C08698=1117.491,408.692,-92.571,-176.642,11.635,149.513
C08699=1117.494,408.445,-92.532,-176.644,11.630,149.512
C08700=1117.498,408.198,-92.493,-176.645,11.625,149.511
C08701=1117.502,407.951,-92.453,-176.646,11.620,149.510
C08702=1117.505,407.705,-92.414,-176.647,11.615,149.509
C08703=1117.508,407.458,-92.375,-176.648,11.611,149.508
C08704=1117.512,407.211,-92.336,-176.650,11.606,149.508
C08705=1117.516,406.963,-92.298,-176.651,11.602,149.507
C08706=1117.519,406.716,-92.258,-176.652,11.596,149.506
C08707=1117.522,406.470,-92.220,-176.653,11.592,149.505
C08708=1117.526,406.223,-92.181,-176.655,11.588,149.504
C08709=1117.530,405.977,-92.142,-176.656,11.583,149.503
C08710=1117.534,405.729,-92.103,-176.658,11.579,149.502
C08711=1117.537,405.482,-92.064,-176.659,11.574,149.501
C08712=1117.540,405.235,-92.025,-176.660,11.570,149.501
C08713=1117.544,404.988,-91.986,-176.662,11.565,149.500
C08714=1117.548,404.741,-91.947,-176.663,11.561,149.499
C08715=1117.551,404.495,-91.909,-176.664,11.557,149.498
C08716=1117.555,404.248,-91.870,-176.666,11.552,149.498
C08717=1117.559,404.001,-91.831,-176.667,11.547,149.497
C08718=1117.562,403.754,-91.793,-176.669,11.543,149.496
C08719=1117.565,403.542,-91.759,-176.670,11.540,149.495
C08720=1117.568,403.330,-91.726,-176.671,11.536,149.495
C08721=1117.571,403.118,-91.693,-176.672,11.533,149.494
C08722=1117.574,402.907,-91.659,-176.674,11.529,149.494
C08723=1117.578,402.695,-91.626,-176.675,11.526,149.493
C08724=1117.581,402.483,-91.593,-176.676,11.522,149.492
C08725=1117.583,402.272,-91.560,-176.677,11.519,149.492
C08726=1117.586,402.060,-91.527,-176.679,11.515,149.491
C08727=1117.590,401.813,-91.488,-176.680,11.511,149.490
C08728=1117.594,401.567,-91.450,-176.682,11.507,149.490
C08729=1117.597,401.320,-91.411,-176.683,11.503,149.489
C08730=1117.601,401.072,-91.372,-176.685,11.499,149.489
C08731=1117.604,400.826,-91.333,-176.686,11.495,149.488
C08732=1117.608,400.578,-91.295,-176.688,11.491,149.487
C08733=1117.612,400.332,-91.256,-176.690,11.488,149.487
C08734=1117.616,400.084,-91.218,-176.691,11.484,149.486
C08735=1117.619,399.837,-91.179,-176.693,11.480,149.486
C08736=1117.622,399.590,-91.141,-176.695,11.476,149.485
C08737=1117.627,399.344,-91.102,-176.697,11.472,149.485
C08738=1117.630,399.097,-91.064,-176.698,11.469,149.484
C08739=1117.633,398.850,-91.025,-176.699,11.466,149.484
C08740=1117.637,398.602,-90.986,-176.701,11.462,149.483
C08741=1117.641,398.356,-90.949,-176.703,11.458,149.482
C08742=1117.645,398.109,-90.910,-176.705,11.454,149.482
C08743=1117.648,397.861,-90.872,-176.707,11.451,149.481
C08744=1117.652,397.615,-90.833,-176.708,11.447,149.481
C08745=1117.655,397.368,-90.795,-176.710,11.444,149.480
C08746=1117.659,397.120,-90.756,-176.712,11.440,149.480
C08747=1117.662,396.874,-90.718,-176.713,11.437,149.479
C08748=1117.667,396.627,-90.679,-176.715,11.433,149.479
C08749=1117.670,396.379,-90.641,-176.717,11.430,149.479
C08750=1117.673,396.132,-90.602,-176.719,11.427,149.478
C08751=1117.677,395.886,-90.565,-176.721,11.423,149.478
C08752=1117.681,395.638,-90.526,-176.722,11.419,149.477
C08753=1117.684,395.391,-90.488,-176.724,11.417,149.477
C08754=1117.689,395.145,-90.449,-176.726,11.413,149.477
C08755=1117.692,394.897,-90.411,-176.728,11.410,149.476
C08756=1117.696,394.650,-90.373,-176.730,11.407,149.476
C08757=1117.699,394.403,-90.335,-176.732,11.404,149.476
C08758=1117.702,394.157,-90.297,-176.733,11.401,149.475
C08759=1117.706,393.909,-90.258,-176.735,11.397,149.475
C08760=1117.710,393.663,-90.220,-176.737,11.394,149.474
C08761=1117.714,393.415,-90.182,-176.739,11.391,149.474
C08762=1117.717,393.168,-90.144,-176.741,11.388,149.474
C08763=1117.721,392.921,-90.105,-176.743,11.386,149.474
C08764=1117.725,392.674,-90.067,-176.745,11.382,149.473
C08765=1117.728,392.428,-90.030,-176.746,11.379,149.473
C08766=1117.732,392.180,-89.991,-176.749,11.376,149.473
C08767=1117.735,391.933,-89.953,-176.750,11.374,149.472
C08768=1117.739,391.686,-89.916,-176.753,11.370,149.472
C08769=1117.743,391.439,-89.877,-176.754,11.368,149.472
C08770=1117.746,391.191,-89.839,-176.757,11.365,149.472
C08771=1117.750,390.945,-89.801,-176.758,11.362,149.471
C08772=1117.754,390.697,-89.763,-176.761,11.359,149.471
C08773=1117.758,390.451,-89.725,-176.763,11.356,149.471
C08774=1117.761,390.203,-89.687,-176.765,11.353,149.471
C08775=1117.764,389.992,-89.654,-176.766,11.351,149.471
C08776=1117.768,389.779,-89.622,-176.768,11.349,149.471
C08777=1117.771,389.569,-89.589,-176.770,11.347,149.470
C08778=1117.774,389.356,-89.557,-176.772,11.344,149.470
C08779=1117.777,389.145,-89.524,-176.774,11.342,149.470
C08780=1117.780,388.932,-89.491,-176.776,11.340,149.470
C08781=1117.783,388.720,-89.459,-176.777,11.337,149.470
C08782=1117.787,388.509,-89.426,-176.779,11.335,149.470
C08783=1117.790,388.262,-89.388,-176.781,11.332,149.470
C08784=1117.793,388.015,-89.351,-176.783,11.330,149.469
C08785=1117.798,387.767,-89.313,-176.786,11.327,149.469
C08786=1117.801,387.520,-89.275,-176.787,11.325,149.469
C08787=1117.805,387.274,-89.238,-176.790,11.323,149.469
C08788=1117.808,387.026,-89.200,-176.792,11.320,149.469
C08789=1117.812,386.780,-89.162,-176.794,11.317,149.469
C08790=1117.816,386.532,-89.124,-176.796,11.315,149.469
C08791=1117.820,386.286,-89.086,-176.798,11.313,149.469
C08792=1117.823,386.038,-89.048,-176.800,11.310,149.469
C08793=1117.827,385.791,-89.011,-176.803,11.307,149.469
C08794=1117.831,385.544,-88.973,-176.805,11.305,149.469
C08795=1117.835,385.297,-88.935,-176.807,11.303,149.469
C08796=1117.838,385.050,-88.897,-176.809,11.301,149.468
C08797=1117.841,384.803,-88.860,-176.811,11.299,149.469
C08798=1117.845,384.555,-88.822,-176.814,11.296,149.469
C08799=1117.849,384.309,-88.785,-176.816,11.294,149.468
C08800=1117.853,384.061,-88.746,-176.818,11.291,149.468
C08801=1117.856,383.814,-88.709,-176.821,11.289,149.468
C08802=1117.860,383.567,-88.671,-176.823,11.287,149.469
C08803=1117.864,383.320,-88.634,-176.826,11.285,149.469
C08804=1117.867,383.073,-88.596,-176.829,11.282,149.469
C08805=1117.871,382.826,-88.559,-176.832,11.279,149.469
C08806=1117.874,382.578,-88.521,-176.835,11.276,149.469
C08807=1117.878,382.332,-88.483,-176.837,11.274,149.469
C08808=1117.882,382.084,-88.446,-176.840,11.272,149.469
C08809=1117.886,381.837,-88.408,-176.843,11.269,149.469
C08810=1117.889,381.590,-88.370,-176.847,11.267,149.469
C08811=1117.893,381.342,-88.333,-176.850,11.264,149.469
C08812=1117.897,381.096,-88.296,-176.853,11.261,149.469
C08813=1117.901,380.848,-88.259,-176.856,11.259,149.470
C08814=1117.904,380.601,-88.221,-176.859,11.256,149.470
C08815=1117.908,380.354,-88.184,-176.862,11.254,149.470
C08816=1117.912,380.107,-88.146,-176.866,11.251,149.470
C08817=1117.915,379.860,-88.109,-176.868,11.248,149.470
C08818=1117.919,379.613,-88.071,-176.872,11.246,149.470
C08819=1117.923,379.366,-88.034,-176.875,11.243,149.470
C08820=1117.926,379.118,-87.997,-176.877,11.241,149.470
C08821=1117.930,378.871,-87.960,-176.881,11.239,149.471
C08822=1117.934,378.624,-87.922,-176.884,11.236,149.471
C08823=1117.938,378.376,-87.885,-176.887,11.233,149.471
C08824=1117.941,378.130,-87.847,-176.890,11.231,149.471
C08825=1117.946,377.883,-87.810,-176.893,11.229,149.471
C08826=1117.949,377.635,-87.773,-176.896,11.226,149.471
C08827=1117.953,377.388,-87.736,-176.900,11.223,149.472
C08828=1117.957,377.141,-87.699,-176.903,11.221,149.472
C08829=1117.960,376.894,-87.661,-176.906,11.218,149.472
C08830=1117.964,376.647,-87.624,-176.909,11.216,149.472
C08831=1117.967,376.435,-87.592,-176.912,11.214,149.472
C08832=1117.971,376.223,-87.561,-176.914,11.212,149.472
C08833=1117.973,376.011,-87.529,-176.917,11.209,149.472
C08834=1117.977,375.798,-87.497,-176.920,11.208,149.473
C08835=1117.980,375.587,-87.465,-176.923,11.206,149.473
C08836=1117.983,375.375,-87.433,-176.926,11.203,149.473
C08837=1117.986,375.163,-87.402,-176.928,11.201,149.473
C08838=1117.990,374.951,-87.369,-176.930,11.199,149.473
C08839=1117.993,374.704,-87.333,-176.934,11.197,149.473
C08840=1117.997,374.456,-87.296,-176.937,11.194,149.474
C08841=1118.001,374.209,-87.258,-176.940,11.192,149.474
C08842=1118.005,373.962,-87.221,-176.944,11.189,149.474
C08843=1118.009,373.715,-87.185,-176.947,11.187,149.474
C08844=1118.012,373.467,-87.148,-176.950,11.184,149.474
C08845=1118.016,373.220,-87.111,-176.954,11.182,149.475
C08846=1118.020,372.973,-87.074,-176.957,11.179,149.475
C08847=1118.024,372.726,-87.037,-176.960,11.178,149.475
C08848=1118.027,372.478,-87.000,-176.963,11.175,149.475
C08849=1118.030,372.232,-86.963,-176.966,11.173,149.476
C08850=1118.034,371.984,-86.926,-176.969,11.170,149.476
C08851=1118.039,371.737,-86.890,-176.973,11.168,149.476
C08852=1118.042,371.489,-86.852,-176.976,11.165,149.476
C08853=1118.045,371.242,-86.816,-176.979,11.163,149.476
C08854=1118.049,370.995,-86.779,-176.983,11.160,149.477
C08855=1118.054,370.748,-86.742,-176.986,11.158,149.477
C08856=1118.057,370.501,-86.706,-176.989,11.155,149.477
C08857=1118.060,370.253,-86.669,-176.993,11.153,149.477
C08858=1118.065,370.006,-86.632,-176.995,11.151,149.477
C08859=1118.068,369.759,-86.596,-176.998,11.149,149.478
C08860=1118.072,369.511,-86.560,-177.002,11.146,149.478
C08861=1118.076,369.264,-86.523,-177.005,11.144,149.478
C08862=1118.079,369.017,-86.486,-177.009,11.142,149.478
C08863=1118.083,368.769,-86.449,-177.012,11.139,149.479
C08864=1118.087,368.522,-86.412,-177.015,11.137,149.479
C08865=1118.091,368.275,-86.376,-177.019,11.134,149.479
C08866=1118.095,368.028,-86.340,-177.022,11.132,149.479
C08867=1118.099,367.780,-86.303,-177.025,11.129,149.479
C08868=1118.103,367.533,-86.267,-177.029,11.127,149.480
C08869=1118.106,367.286,-86.230,-177.032,11.124,149.480
C08870=1118.109,367.039,-86.193,-177.036,11.122,149.480
C08871=1118.114,366.791,-86.157,-177.038,11.121,149.481
C08872=1118.117,366.544,-86.121,-177.042,11.118,149.481
C08873=1118.121,366.297,-86.084,-177.045,11.116,149.481
C08874=1118.125,366.050,-86.047,-177.048,11.113,149.481
C08875=1118.129,365.802,-86.012,-177.051,11.111,149.481
C08876=1118.133,365.555,-85.975,-177.055,11.108,149.482
C08877=1118.136,365.308,-85.939,-177.058,11.106,149.482
C08878=1118.141,365.060,-85.902,-177.062,11.104,149.482
C08879=1118.144,364.813,-85.866,-177.065,11.101,149.482
C08880=1118.148,364.565,-85.830,-177.068,11.099,149.483
C08881=1118.151,364.318,-85.793,-177.072,11.096,149.483
C08882=1118.155,364.071,-85.756,-177.075,11.094,149.483
C08883=1118.159,363.823,-85.721,-177.079,11.092,149.483
C08884=1118.162,363.576,-85.685,-177.082,11.089,149.484
C08885=1118.167,363.329,-85.649,-177.085,11.087,149.484
C08886=1118.170,363.082,-85.612,-177.089,11.084,149.484
C08887=1118.174,362.870,-85.581,-177.091,11.082,149.484
C08888=1118.177,362.657,-85.550,-177.095,11.080,149.485
C08889=1118.181,362.445,-85.519,-177.097,11.078,149.485
C08890=1118.184,362.233,-85.488,-177.100,11.077,149.485
C08891=1118.187,362.021,-85.458,-177.103,11.074,149.485
C08892=1118.190,361.809,-85.427,-177.106,11.072,149.486
C08893=1118.193,361.596,-85.395,-177.109,11.070,149.486
C08894=1118.197,361.384,-85.365,-177.112,11.068,149.486
C08895=1118.200,361.137,-85.328,-177.115,11.066,149.486
C08896=1118.204,360.890,-85.293,-177.118,11.063,149.486
C08897=1118.208,360.643,-85.256,-177.122,11.061,149.487
C08898=1118.212,360.395,-85.220,-177.125,11.059,149.487
C08899=1118.215,360.148,-85.185,-177.129,11.056,149.487
C08900=1118.219,359.901,-85.148,-177.132,11.054,149.487
C08901=1118.223,359.653,-85.112,-177.135,11.051,149.488
C08902=1118.227,359.406,-85.077,-177.139,11.049,149.488
C08903=1118.231,359.158,-85.041,-177.142,11.047,149.488
C08904=1118.234,358.911,-85.004,-177.146,11.044,149.489
C08905=1118.238,358.663,-84.969,-177.149,11.042,149.489
C08906=1118.242,358.416,-84.933,-177.152,11.039,149.489
C08907=1118.246,358.169,-84.896,-177.156,11.037,149.489
C08908=1118.250,357.921,-84.861,-177.159,11.035,149.490
C08909=1118.253,357.674,-84.825,-177.163,11.032,149.490
C08910=1118.257,357.426,-84.790,-177.166,11.030,149.490
C08911=1118.261,357.179,-84.755,-177.169,11.027,149.490
C08912=1118.266,356.932,-84.718,-177.173,11.025,149.491
C08913=1118.269,356.685,-84.682,-177.176,11.023,149.491
C08914=1118.273,356.437,-84.647,-177.180,11.020,149.491
C08915=1118.276,356.190,-84.611,-177.183,11.018,149.491
C08916=1118.280,355.942,-84.576,-177.186,11.015,149.492
C08917=1118.284,355.694,-84.539,-177.191,11.012,149.492
C08918=1118.288,355.447,-84.504,-177.194,11.010,149.492
C08919=1118.292,355.199,-84.468,-177.197,11.007,149.492
C08920=1118.296,354.953,-84.433,-177.200,11.005,149.493
C08921=1118.300,354.705,-84.398,-177.204,11.002,149.493
C08922=1118.303,354.458,-84.362,-177.207,11.000,149.493
C08923=1118.307,354.210,-84.326,-177.211,10.998,149.493
C08924=1118.311,353.963,-84.291,-177.214,10.995,149.494
C08925=1118.315,353.715,-84.255,-177.217,10.993,149.494
C08926=1118.319,353.468,-84.220,-177.221,10.991,149.494
C08927=1118.323,353.220,-84.184,-177.224,10.988,149.494
C08928=1118.327,352.973,-84.149,-177.228,10.985,149.495
C08929=1118.330,352.725,-84.113,-177.232,10.983,149.495
C08930=1118.334,352.478,-84.077,-177.235,10.980,149.495
C08931=1118.338,352.231,-84.042,-177.238,10.978,149.495
C08932=1118.342,351.983,-84.007,-177.242,10.975,149.496
C08933=1118.346,351.736,-83.972,-177.245,10.973,149.496
C08934=1118.349,351.488,-83.936,-177.248,10.970,149.496
C08935=1118.353,351.241,-83.901,-177.252,10.968,149.496
C08936=1118.357,350.994,-83.866,-177.255,10.965,149.496
C08937=1118.361,350.746,-83.831,-177.259,10.962,149.497
C08938=1118.365,350.498,-83.795,-177.262,10.960,149.497
C08939=1118.369,350.251,-83.760,-177.266,10.958,149.497
C08940=1118.373,350.004,-83.724,-177.269,10.955,149.498
C08941=1118.377,349.756,-83.690,-177.272,10.953,149.498
C08942=1118.381,349.508,-83.654,-177.276,10.949,149.498
C08943=1118.384,349.296,-83.624,-177.279,10.947,149.498
C08944=1118.387,349.084,-83.594,-177.281,10.946,149.498
C08945=1118.391,348.872,-83.564,-177.285,10.943,149.499
C08946=1118.395,348.659,-83.534,-177.287,10.941,149.499
C08947=1118.397,348.447,-83.503,-177.290,10.940,149.499
C08948=1118.400,348.235,-83.474,-177.293,10.937,149.499
C08949=1118.404,348.022,-83.443,-177.295,10.935,149.499
C08950=1118.407,347.810,-83.413,-177.299,10.933,149.499
C08951=1118.411,347.562,-83.378,-177.301,10.931,149.499
C08952=1118.415,347.316,-83.343,-177.304,10.928,149.500
C08953=1118.419,347.067,-83.308,-177.307,10.926,149.500
C08954=1118.423,346.820,-83.273,-177.311,10.923,149.500
C08955=1118.427,346.573,-83.239,-177.314,10.921,149.500
C08956=1118.430,346.325,-83.203,-177.317,10.918,149.501
C08957=1118.434,346.077,-83.168,-177.320,10.916,149.501
C08958=1118.439,345.830,-83.133,-177.324,10.913,149.501
C08959=1118.442,345.582,-83.098,-177.327,10.911,149.501
C08960=1118.447,345.335,-83.063,-177.330,10.908,149.501
C08961=1118.450,345.088,-83.029,-177.334,10.906,149.502
C08962=1118.454,344.840,-82.993,-177.337,10.903,149.502
C08963=1118.458,344.593,-82.959,-177.340,10.900,149.502
C08964=1118.462,344.345,-82.924,-177.343,10.898,149.502
C08965=1118.465,344.097,-82.889,-177.346,10.896,149.502
C08966=1118.470,343.850,-82.855,-177.349,10.894,149.503
C08967=1118.473,343.602,-82.819,-177.352,10.891,149.503
C08968=1118.478,343.355,-82.785,-177.356,10.889,149.503
C08969=1118.481,343.107,-82.750,-177.359,10.886,149.503
C08970=1118.486,342.860,-82.716,-177.362,10.884,149.503
C08971=1118.489,342.612,-82.680,-177.365,10.881,149.504
C08972=1118.493,342.364,-82.646,-177.369,10.879,149.504
C08973=1118.497,342.117,-82.612,-177.372,10.876,149.504
C08974=1118.501,341.870,-82.576,-177.375,10.874,149.504
C08975=1118.505,341.622,-82.542,-177.378,10.871,149.504
C08976=1118.509,341.374,-82.507,-177.381,10.869,149.505
C08977=1118.513,341.127,-82.473,-177.385,10.866,149.505
C08978=1118.517,340.879,-82.438,-177.387,10.865,149.505
C08979=1118.521,340.632,-82.404,-177.390,10.862,149.505
C08980=1118.525,340.384,-82.369,-177.394,10.859,149.505
C08981=1118.529,340.137,-82.334,-177.397,10.857,149.506
C08982=1118.532,339.889,-82.300,-177.400,10.854,149.506
C08983=1118.537,339.642,-82.266,-177.403,10.852,149.506
C08984=1118.540,339.394,-82.231,-177.407,10.849,149.506
C08985=1118.545,339.146,-82.197,-177.410,10.847,149.506
C08986=1118.549,338.898,-82.162,-177.413,10.844,149.507
C08987=1118.553,338.651,-82.128,-177.416,10.842,149.507
C08988=1118.557,338.403,-82.093,-177.419,10.839,149.507
C08989=1118.560,338.157,-82.059,-177.423,10.837,149.507
C08990=1118.564,337.908,-82.024,-177.426,10.834,149.507
C08991=1118.568,337.661,-81.990,-177.429,10.832,149.508
C08992=1118.572,337.413,-81.955,-177.432,10.830,149.508
C08993=1118.576,337.166,-81.921,-177.435,10.827,149.508
C08994=1118.580,336.917,-81.887,-177.438,10.825,149.508
C08995=1118.584,336.670,-81.853,-177.442,10.822,149.508
C08996=1118.588,336.423,-81.819,-177.444,10.819,149.508
C08997=1118.592,336.175,-81.785,-177.448,10.817,149.509
C08998=1118.596,335.928,-81.750,-177.451,10.815,149.509
C08999=1118.599,335.715,-81.721,-177.453,10.813,149.509
C09000=1118.603,335.503,-81.691,-177.457,10.810,149.509
C09001=1118.606,335.290,-81.662,-177.459,10.808,149.509
C09002=1118.609,335.078,-81.632,-177.462,10.806,149.510
C09003=1118.613,334.865,-81.604,-177.465,10.804,149.510
C09004=1118.616,334.653,-81.574,-177.467,10.802,149.510
C09005=1118.619,334.441,-81.544,-177.470,10.799,149.510
C09006=1118.623,334.228,-81.516,-177.473,10.798,149.510
C09007=1118.627,333.981,-81.482,-177.476,10.795,149.510
C09008=1118.631,333.733,-81.448,-177.479,10.792,149.510
C09009=1118.634,333.485,-81.413,-177.482,10.790,149.511
C09010=1118.639,333.238,-81.380,-177.486,10.787,149.511
C09011=1118.643,332.989,-81.345,-177.489,10.785,149.511
C09012=1118.646,332.742,-81.311,-177.491,10.783,149.511
C09013=1118.650,332.495,-81.277,-177.495,10.780,149.512
C09014=1118.655,332.246,-81.243,-177.498,10.778,149.512
C09015=1118.658,331.999,-81.209,-177.501,10.775,149.512
C09016=1118.662,331.752,-81.175,-177.504,10.773,149.512
C09017=1118.666,331.504,-81.141,-177.508,10.770,149.512
C09018=1118.670,331.256,-81.107,-177.511,10.768,149.513
C09019=1118.674,331.009,-81.073,-177.514,10.765,149.513
C09020=1118.678,330.761,-81.040,-177.517,10.763,149.513
C09021=1118.682,330.513,-81.005,-177.520,10.760,149.513
C09022=1118.686,330.266,-80.972,-177.523,10.757,149.513
C09023=1118.690,330.018,-80.938,-177.527,10.755,149.513
C09024=1118.694,329.770,-80.905,-177.530,10.753,149.514
C09025=1118.698,329.523,-80.870,-177.533,10.751,149.514
C09026=1118.702,329.275,-80.837,-177.536,10.748,149.514
C09027=1118.706,329.027,-80.803,-177.539,10.746,149.514
C09028=1118.710,328.780,-80.769,-177.542,10.743,149.514
C09029=1118.714,328.532,-80.736,-177.545,10.740,149.515
C09030=1118.718,328.284,-80.702,-177.549,10.738,149.515
C09031=1118.722,328.037,-80.668,-177.552,10.736,149.515
C09032=1118.726,327.789,-80.635,-177.555,10.733,149.515
C09033=1118.730,327.542,-80.601,-177.558,10.730,149.515
C09034=1118.733,327.293,-80.568,-177.561,10.728,149.516
C09035=1118.738,327.046,-80.533,-177.564,10.725,149.516
C09036=1118.742,326.798,-80.500,-177.568,10.723,149.516
C09037=1118.746,326.550,-80.467,-177.571,10.720,149.516
C09038=1118.750,326.303,-80.433,-177.573,10.718,149.516
C09039=1118.753,326.055,-80.399,-177.577,10.716,149.516
C09040=1118.758,325.807,-80.366,-177.580,10.713,149.517
C09041=1118.761,325.560,-80.332,-177.583,10.710,149.517
C09042=1118.766,325.312,-80.299,-177.586,10.708,149.517
C09043=1118.769,325.064,-80.266,-177.589,10.706,149.517
C09044=1118.773,324.816,-80.232,-177.592,10.703,149.517
C09045=1118.777,324.569,-80.199,-177.596,10.700,149.518
C09046=1118.782,324.321,-80.165,-177.599,10.698,149.518
C09047=1118.786,324.073,-80.132,-177.602,10.695,149.518
C09048=1118.790,323.826,-80.099,-177.605,10.693,149.518
C09049=1118.793,323.578,-80.064,-177.609,10.690,149.518
C09050=1118.798,323.330,-80.031,-177.612,10.687,149.518
C09051=1118.802,323.082,-79.998,-177.614,10.686,149.519
C09052=1118.806,322.835,-79.965,-177.618,10.683,149.519
C09053=1118.810,322.587,-79.932,-177.621,10.681,149.519
C09054=1118.814,322.339,-79.899,-177.624,10.678,149.519
C09055=1118.817,322.126,-79.870,-177.627,10.675,149.519
C09056=1118.820,321.914,-79.841,-177.629,10.674,149.520
C09057=1118.823,321.701,-79.813,-177.632,10.672,149.520
C09058=1118.827,321.489,-79.785,-177.635,10.669,149.520
C09059=1118.831,321.276,-79.756,-177.637,10.667,149.520
C09060=1118.834,321.063,-79.727,-177.640,10.665,149.520
C09061=1118.838,320.851,-79.699,-177.643,10.663,149.520
C09062=1118.841,320.639,-79.671,-177.645,10.661,149.520
C09063=1118.845,320.391,-79.637,-177.649,10.658,149.521
C09064=1118.849,320.143,-79.604,-177.652,10.656,149.521
C09065=1118.853,319.896,-79.571,-177.655,10.653,149.521
C09066=1118.857,319.648,-79.538,-177.658,10.651,149.521
C09067=1118.861,319.400,-79.505,-177.661,10.648,149.521
C09068=1118.864,319.152,-79.472,-177.664,10.646,149.522
C09069=1118.868,318.904,-79.439,-177.668,10.643,149.522
C09070=1118.872,318.656,-79.406,-177.670,10.641,149.522
C09071=1118.876,318.409,-79.372,-177.673,10.639,149.522
C09072=1118.881,318.161,-79.339,-177.676,10.636,149.522
C09073=1118.885,317.913,-79.307,-177.680,10.633,149.523
C09074=1118.888,317.665,-79.274,-177.683,10.631,149.523
C09075=1118.893,317.418,-79.241,-177.686,10.628,149.523
C09076=1118.897,317.170,-79.208,-177.689,10.626,149.523
C09077=1118.901,316.922,-79.175,-177.693,10.623,149.523
C09078=1118.905,316.674,-79.142,-177.695,10.621,149.523
C09079=1118.909,316.426,-79.110,-177.699,10.618,149.524
C09080=1118.913,316.179,-79.077,-177.702,10.615,149.524
C09081=1118.917,315.931,-79.043,-177.705,10.613,149.524
C09082=1118.921,315.683,-79.010,-177.708,10.610,149.524
C09083=1118.925,315.435,-78.978,-177.711,10.608,149.524
C09084=1118.929,315.187,-78.945,-177.714,10.606,149.525
C09085=1118.933,314.940,-78.912,-177.717,10.603,149.525
C09086=1118.937,314.692,-78.880,-177.720,10.601,149.525
C09087=1118.941,314.444,-78.847,-177.724,10.598,149.525
C09088=1118.945,314.196,-78.814,-177.726,10.596,149.525
C09089=1118.949,313.948,-78.782,-177.730,10.593,149.526
C09090=1118.953,313.700,-78.749,-177.733,10.590,149.526
C09091=1118.957,313.453,-78.716,-177.736,10.588,149.526
C09092=1118.961,313.205,-78.684,-177.739,10.585,149.526
C09093=1118.965,312.957,-78.651,-177.742,10.583,149.526
C09094=1118.969,312.709,-78.618,-177.746,10.580,149.526
C09095=1118.973,312.461,-78.586,-177.748,10.578,149.527
C09096=1118.978,312.214,-78.553,-177.751,10.576,149.527
C09097=1118.982,311.966,-78.521,-177.754,10.573,149.527
C09098=1118.985,311.718,-78.488,-177.758,10.571,149.527
C09099=1118.990,311.470,-78.456,-177.761,10.568,149.527
C09100=1118.993,311.223,-78.423,-177.764,10.565,149.527
C09101=1118.998,310.974,-78.391,-177.767,10.563,149.528
C09102=1119.001,310.727,-78.358,-177.770,10.560,149.528
C09103=1119.005,310.478,-78.326,-177.773,10.558,149.528
C09104=1119.010,310.230,-78.293,-177.776,10.555,149.528
C09105=1119.014,309.983,-78.261,-177.780,10.553,149.528
C09106=1119.018,309.735,-78.229,-177.782,10.551,149.528
C09107=1119.022,309.488,-78.196,-177.785,10.548,149.529
C09108=1119.026,309.239,-78.164,-177.789,10.546,149.529
C09109=1119.030,308.991,-78.132,-177.792,10.543,149.529
C09110=1119.034,308.743,-78.099,-177.795,10.540,149.529
C09111=1119.038,308.531,-78.071,-177.797,10.539,149.529
C09112=1119.041,308.318,-78.044,-177.800,10.536,149.529
C09113=1119.044,308.106,-78.016,-177.803,10.534,149.530
C09114=1119.048,307.892,-77.988,-177.806,10.531,149.530
C09115=1119.052,307.680,-77.960,-177.808,10.529,149.530
C09116=1119.055,307.467,-77.933,-177.811,10.528,149.530
C09117=1119.058,307.255,-77.905,-177.814,10.525,149.530
C09118=1119.062,307.042,-77.878,-177.816,10.523,149.530
